	//dosilanie
	IF "DB10_instance_SCADA".actDTL_RechargingOn.HOUR < 0
	  OR "DB10_instance_SCADA".actDTL_RechargingOn.HOUR > 23
	  OR "dbHold_Sending".data."Time".Start_dosilanie_1.HOUR < 0
	  OR "dbHold_Sending".data."Time".Start_dosilanie_1.HOUR > 23
	THEN
	  // wypełnij zerami
	  "DB10_instance_SCADA".actDTL_RechargingOn.HOUR := 0;
	  "tempdbHold_SendingTCP".Start_dosilanie_1.HOUR := 0;
	  "dbHold_Sending".data."Time".Start_dosilanie_1.HOUR := 0;
	  ;
	END_IF;
	
	IF "DB10_instance_SCADA".actDTL_RechargingOn.MINUTE < 0
	  OR "DB10_instance_SCADA".actDTL_RechargingOn.MINUTE > 60
	  OR "dbHold_Sending".data."Time".Start_dosilanie_1.MINUTE < 0
	  OR "dbHold_Sending".data."Time".Start_dosilanie_1.MINUTE > 60
	THEN
	  // wypełnij zerami
	  "DB10_instance_SCADA".actDTL_RechargingOn.MINUTE := 0;
	  "tempdbHold_SendingTCP".Start_dosilanie_1.MINUTE := 0;
	  "dbHold_Sending".data."Time".Start_dosilanie_1.MINUTE := 0;
	  ;
	END_IF;
	
	// stop dosilanie
	IF "DB10_instance_SCADA".actDTL_RechargingOff.HOUR < 0
	  OR "DB10_instance_SCADA".actDTL_RechargingOff.HOUR > 23
	  OR "dbHold_Sending".data."Time".Stop_dosilanie_1.HOUR < 0
	  OR "dbHold_Sending".data."Time".Stop_dosilanie_1.HOUR > 23
	THEN
	  // wypełnij zerami
	  "DB10_instance_SCADA".actDTL_RechargingOff.HOUR := 0;
	  "tempdbHold_SendingTCP".Stop_dosilanie_1.HOUR := 0;
	  "dbHold_Sending".data."Time".Stop_dosilanie_1.HOUR := 0;
	  ;
	END_IF;
	
	IF "DB10_instance_SCADA".actDTL_RechargingOff.MINUTE < 0
	  OR "DB10_instance_SCADA".actDTL_RechargingOff.MINUTE > 60
	  OR "dbHold_Sending".data."Time".Stop_dosilanie_1.MINUTE < 0
	  OR "dbHold_Sending".data."Time".Stop_dosilanie_1.MINUTE > 60
	THEN
	  // wypełnij zerami
	  "DB10_instance_SCADA".actDTL_RechargingOff.MINUTE := 0;
	  "tempdbHold_SendingTCP".Stop_dosilanie_1.MINUTE := 0;
	  "dbHold_Sending".data."Time".Stop_dosilanie_1.MINUTE := 0;
	  ;
	END_IF;
	
	
	
	
	
	
	
END_FUNCTION

FUNCTION "Read_MPP04_2_ModbusRTU" : Void   // FC24, LAD
TITLE = Odczyt parametrów z MPP04 Pompownia / Read data from SC100
{ S7_Optimized_Access := 'TRUE' }
AUTHOR : rtecmer
VERSION : 0.1
// Czytanie z przepływomierza pompownia główna. Modbus RTU 19200, bit stop-1, parti-no
// Czytanie z SC1000 
// Obsługa protokołu Master Modbus RTU.  Odczyt pomiarów  i status czujnika SC1000
// stored: AutoNumber false, IsIECCheckEnabled false, SetENOAutomatically false, UDAEnableTagReadback false
   VAR_TEMP
      Wielkość_przeływu_Adres0_0 : DWord;
      Wielkość_przeływu_Adres0_1 : DWord;
      Wielkość_przeływu_Adres2_0 : DWord;
      Wielkość_przeływu_Adres2_2 : DWord;
   END_VAR
   VAR_TEMP   // added for the SCL form of the ladder/FBD networks
      _w1 : Bool;
      _w2 : Bool;
   END_VAR
BEGIN

REGION Network 1: Odczyt parametrów z MPP04 Studnia na tłocznym
   // Czytanie z przepływomierza pompownia główna. Modbus RTU 19200, bit stop-1, parti-no
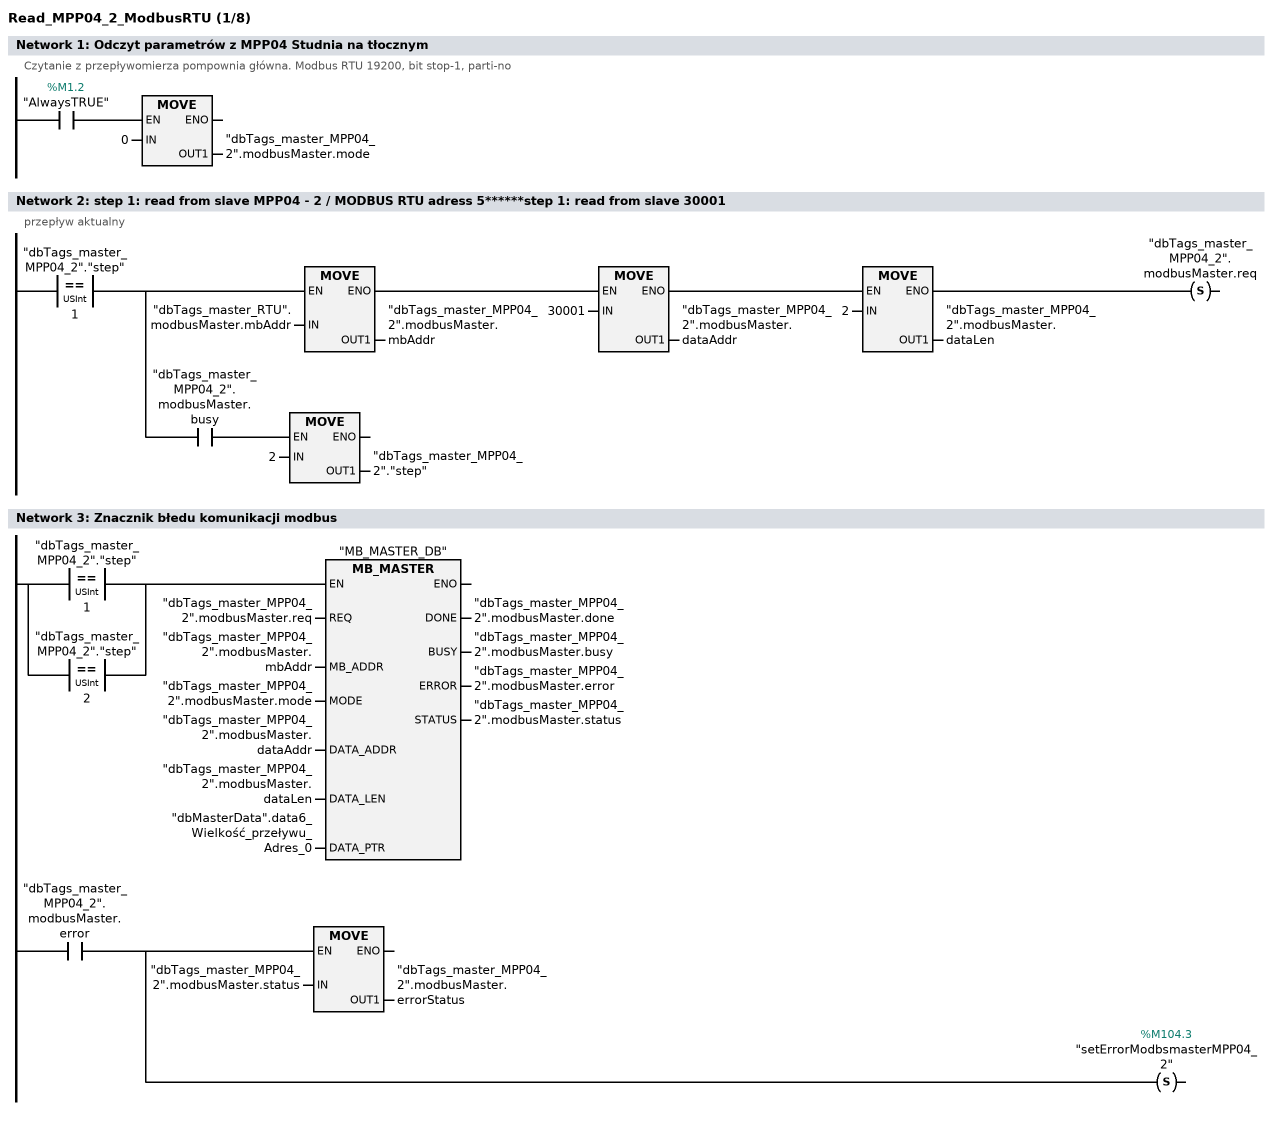
   RUNG wire#powerrail
      Contact( "AlwaysTRUE" )
      { S7_GenerateENO := "TRUE" } Move(in := 0, out1 => "dbTags_master_MPP04_2".modbusMaster.mode)
   END_RUNG
   // the same network as SCL:
   IF "AlwaysTRUE" THEN "dbTags_master_MPP04_2".modbusMaster.mode := 0; END_IF;
END_REGION

REGION Network 2: step 1: read from slave MPP04 - 2 / MODBUS RTU adress 5******step 1: read from slave 30001
   // przepływ aktualny
   RUNG wire#powerrail
      { S7_Templates := "SrcType := USInt" } EQ_Contact(in1 := "dbTags_master_MPP04_2"."step", in2 := 1)
      wire#w1
      Move(in := "dbTags_master_RTU".modbusMaster.mbAddr, out1 => "dbTags_master_MPP04_2".modbusMaster.mbAddr)
      { S7_GenerateENO := "TRUE" } Move(in := 30001, out1 => "dbTags_master_MPP04_2".modbusMaster.dataAddr)
      Move(in := 2, out1 => "dbTags_master_MPP04_2".modbusMaster.dataLen)
      S_Coil( "dbTags_master_MPP04_2".modbusMaster.req )
   END_RUNG
   RUNG wire#w1
      Contact( "dbTags_master_MPP04_2".modbusMaster.busy )
      { S7_GenerateENO := "TRUE" } Move(in := 2, out1 => "dbTags_master_MPP04_2"."step")
   END_RUNG
   // the same network as SCL:
   // ENO of a box is taken as its EN; it also drops when the box reports an error
   #_w1 := "dbTags_master_MPP04_2"."step" = 1;
   IF #_w1 THEN
       "dbTags_master_MPP04_2".modbusMaster.mbAddr := "dbTags_master_RTU".modbusMaster.mbAddr;
       "dbTags_master_MPP04_2".modbusMaster.dataAddr := 30001;
       "dbTags_master_MPP04_2".modbusMaster.dataLen := 2;
       "dbTags_master_MPP04_2".modbusMaster.req := TRUE;
   END_IF;
   IF #_w1 AND "dbTags_master_MPP04_2".modbusMaster.busy THEN "dbTags_master_MPP04_2"."step" := 2; END_IF;
END_REGION

REGION Network 3: Znacznik błedu komunikacji modbus
   RUNG wire#powerrail
      { S7_Templates := "SrcType := USInt" } EQ_Contact(in1 := "dbTags_master_MPP04_2"."step", in2 := 1)
      wire#w1
      "MB_MASTER_DB".MB_MASTER(REQ := "dbTags_master_MPP04_2".modbusMaster.req, MB_ADDR := "dbTags_master_MPP04_2".modbusMaster.mbAddr, MODE := "dbTags_master_MPP04_2".modbusMaster.mode, DATA_ADDR := "dbTags_master_MPP04_2".modbusMaster.dataAddr, DATA_LEN := "dbTags_master_MPP04_2".modbusMaster.dataLen, DATA_PTR := "dbMasterData".data6_Wielkość_przeływu_Adres_0, DONE => "dbTags_master_MPP04_2".modbusMaster.done, BUSY => "dbTags_master_MPP04_2".modbusMaster.busy, ERROR => "dbTags_master_MPP04_2".modbusMaster.error, STATUS => "dbTags_master_MPP04_2".modbusMaster.status)
   END_RUNG
   RUNG wire#powerrail
      { S7_Templates := "SrcType := USInt" } EQ_Contact(in1 := "dbTags_master_MPP04_2"."step", in2 := 2)
   END_RUNG wire#w1
   RUNG wire#powerrail
      Contact( "dbTags_master_MPP04_2".modbusMaster.error )
      wire#w2
      { S7_GenerateENO := "TRUE" } Move(in := "dbTags_master_MPP04_2".modbusMaster.status, out1 => "dbTags_master_MPP04_2".modbusMaster.errorStatus)
   END_RUNG
   RUNG wire#w2
      S_Coil( "setErrorModbsmasterMPP04_2" )
   END_RUNG
   // the same network as SCL:
   IF ("dbTags_master_MPP04_2"."step" = 1) OR ("dbTags_master_MPP04_2"."step" = 2) THEN
       "MB_MASTER_DB"(REQ := "dbTags_master_MPP04_2".modbusMaster.req,   // MB_MASTER
                      MB_ADDR := "dbTags_master_MPP04_2".modbusMaster.mbAddr,
                      MODE := "dbTags_master_MPP04_2".modbusMaster.mode,
                      DATA_ADDR := "dbTags_master_MPP04_2".modbusMaster.dataAddr,
                      DATA_LEN := "dbTags_master_MPP04_2".modbusMaster.dataLen,
                      DATA_PTR := "dbMasterData".data6_Wielkość_przeływu_Adres_0,
                      DONE => "dbTags_master_MPP04_2".modbusMaster.done,
                      BUSY => "dbTags_master_MPP04_2".modbusMaster.busy,
                      ERROR => "dbTags_master_MPP04_2".modbusMaster.error,
                      STATUS => "dbTags_master_MPP04_2".modbusMaster.status);
   END_IF;
   IF "dbTags_master_MPP04_2".modbusMaster.error THEN
       "dbTags_master_MPP04_2".modbusMaster.errorStatus := "dbTags_master_MPP04_2".modbusMaster.status;
       "setErrorModbsmasterMPP04_2" := TRUE;
   END_IF;
END_REGION

REGION Network 4: step 4: save received data / step 2: save received data 30001
   // Pomiar Temperatury KDN1
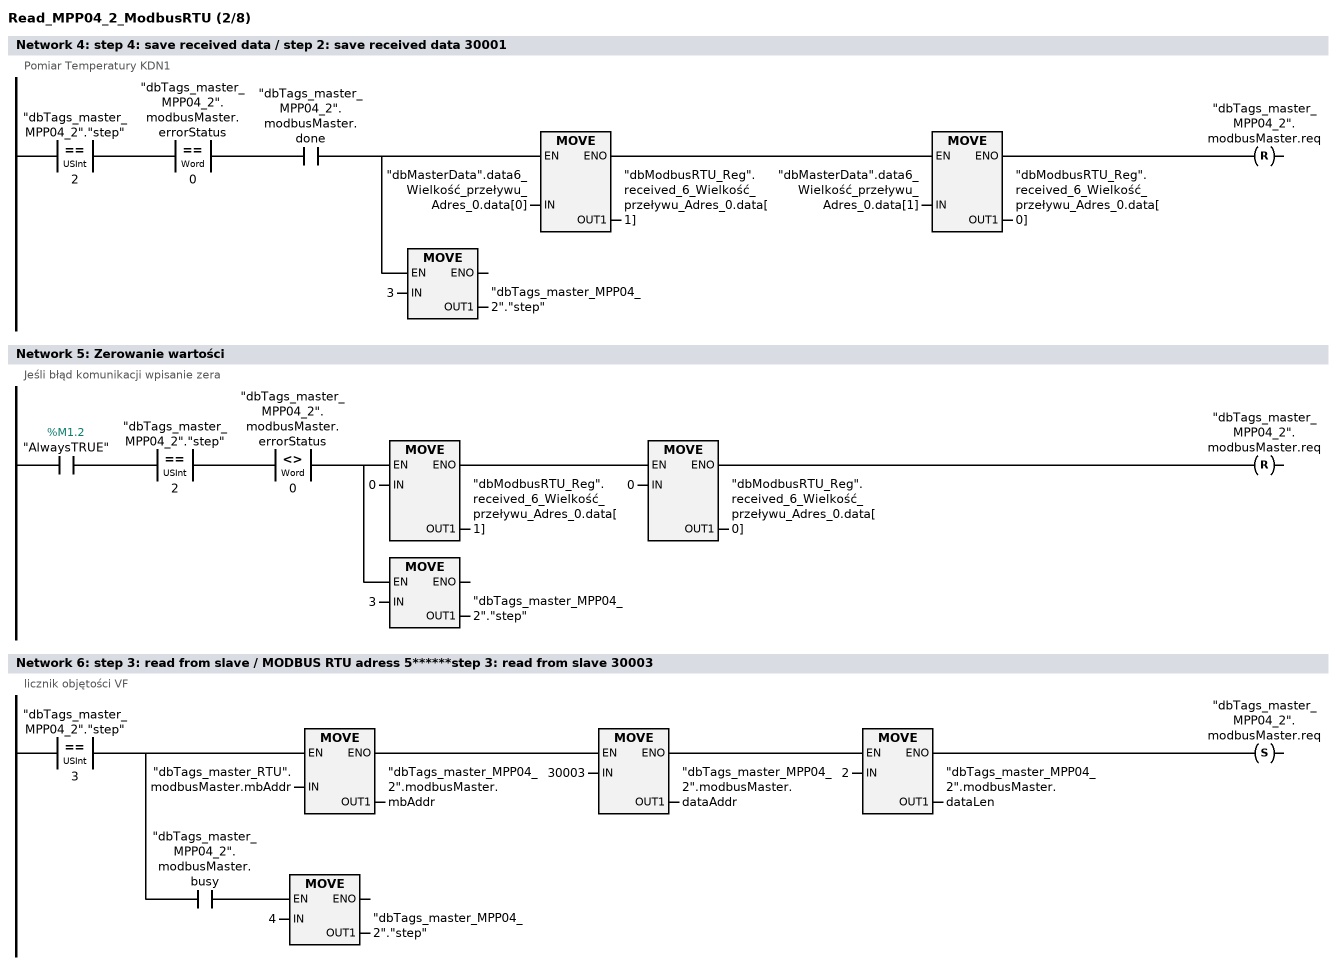
   RUNG wire#powerrail
      { S7_Templates := "SrcType := USInt" } EQ_Contact(in1 := "dbTags_master_MPP04_2"."step", in2 := 2)
      { S7_Templates := "SrcType := Word" } EQ_Contact(in1 := "dbTags_master_MPP04_2".modbusMaster.errorStatus, in2 := 0)
      Contact( "dbTags_master_MPP04_2".modbusMaster.done )
      wire#w1
      { S7_GenerateENO := "TRUE" } Move(in := "dbMasterData".data6_Wielkość_przeływu_Adres_0.data[0], out1 => "dbModbusRTU_Reg".received_6_Wielkość_przeływu_Adres_0.data[1])
      { S7_GenerateENO := "TRUE" } Move(in := "dbMasterData".data6_Wielkość_przeływu_Adres_0.data[1], out1 => "dbModbusRTU_Reg".received_6_Wielkość_przeływu_Adres_0.data[0])
      R_Coil( "dbTags_master_MPP04_2".modbusMaster.req )
   END_RUNG
   RUNG wire#w1
      { S7_GenerateENO := "TRUE" } Move(in := 3, out1 => "dbTags_master_MPP04_2"."step")
   END_RUNG
   // the same network as SCL:
   // ENO of a box is taken as its EN; it also drops when the box reports an error
   IF ("dbTags_master_MPP04_2"."step" = 2) AND ("dbTags_master_MPP04_2".modbusMaster.errorStatus = 0) AND "dbTags_master_MPP04_2".modbusMaster.done THEN
       "dbModbusRTU_Reg".received_6_Wielkość_przeływu_Adres_0.data[1] := "dbMasterData".data6_Wielkość_przeływu_Adres_0.data[0];
       "dbModbusRTU_Reg".received_6_Wielkość_przeływu_Adres_0.data[0] := "dbMasterData".data6_Wielkość_przeływu_Adres_0.data[1];
       "dbTags_master_MPP04_2".modbusMaster.req := FALSE;
       "dbTags_master_MPP04_2"."step" := 3;
   END_IF;
END_REGION

REGION Network 5: Zerowanie wartości
   // Jeśli błąd komunikacji wpisanie zera
   RUNG wire#powerrail
      Contact( "AlwaysTRUE" )
      { S7_Templates := "SrcType := USInt" } EQ_Contact(in1 := "dbTags_master_MPP04_2"."step", in2 := 2)
      { S7_Templates := "SrcType := Word" } NE_Contact(in1 := "dbTags_master_MPP04_2".modbusMaster.errorStatus, in2 := 0)
      wire#w1
      { S7_GenerateENO := "TRUE" } Move(in := 0, out1 => "dbModbusRTU_Reg".received_6_Wielkość_przeływu_Adres_0.data[1])
      { S7_GenerateENO := "TRUE" } Move(in := 0, out1 => "dbModbusRTU_Reg".received_6_Wielkość_przeływu_Adres_0.data[0])
      R_Coil( "dbTags_master_MPP04_2".modbusMaster.req )
   END_RUNG
   RUNG wire#w1
      { S7_GenerateENO := "TRUE" } Move(in := 3, out1 => "dbTags_master_MPP04_2"."step")
   END_RUNG
   // the same network as SCL:
   // ENO of a box is taken as its EN; it also drops when the box reports an error
   IF "AlwaysTRUE" AND ("dbTags_master_MPP04_2"."step" = 2) AND ("dbTags_master_MPP04_2".modbusMaster.errorStatus <> 0) THEN
       "dbModbusRTU_Reg".received_6_Wielkość_przeływu_Adres_0.data[1] := 0;
       "dbModbusRTU_Reg".received_6_Wielkość_przeływu_Adres_0.data[0] := 0;
       "dbTags_master_MPP04_2".modbusMaster.req := FALSE;
       "dbTags_master_MPP04_2"."step" := 3;
   END_IF;
END_REGION

REGION Network 6: step 3: read from slave / MODBUS RTU adress 5******step 3: read from slave 30003
   // licznik objętości VF
   RUNG wire#powerrail
      { S7_Templates := "SrcType := USInt" } EQ_Contact(in1 := "dbTags_master_MPP04_2"."step", in2 := 3)
      wire#w1
      Move(in := "dbTags_master_RTU".modbusMaster.mbAddr, out1 => "dbTags_master_MPP04_2".modbusMaster.mbAddr)
      { S7_GenerateENO := "TRUE" } Move(in := 30003, out1 => "dbTags_master_MPP04_2".modbusMaster.dataAddr)
      Move(in := 2, out1 => "dbTags_master_MPP04_2".modbusMaster.dataLen)
      S_Coil( "dbTags_master_MPP04_2".modbusMaster.req )
   END_RUNG
   RUNG wire#w1
      Contact( "dbTags_master_MPP04_2".modbusMaster.busy )
      { S7_GenerateENO := "TRUE" } Move(in := 4, out1 => "dbTags_master_MPP04_2"."step")
   END_RUNG
   // the same network as SCL:
   // ENO of a box is taken as its EN; it also drops when the box reports an error
   #_w1 := "dbTags_master_MPP04_2"."step" = 3;
   IF #_w1 THEN
       "dbTags_master_MPP04_2".modbusMaster.mbAddr := "dbTags_master_RTU".modbusMaster.mbAddr;
       "dbTags_master_MPP04_2".modbusMaster.dataAddr := 30003;
       "dbTags_master_MPP04_2".modbusMaster.dataLen := 2;
       "dbTags_master_MPP04_2".modbusMaster.req := TRUE;
   END_IF;
   IF #_w1 AND "dbTags_master_MPP04_2".modbusMaster.busy THEN "dbTags_master_MPP04_2"."step" := 4; END_IF;
END_REGION

REGION Network 7: Znacznik błedu komunikacji modbus
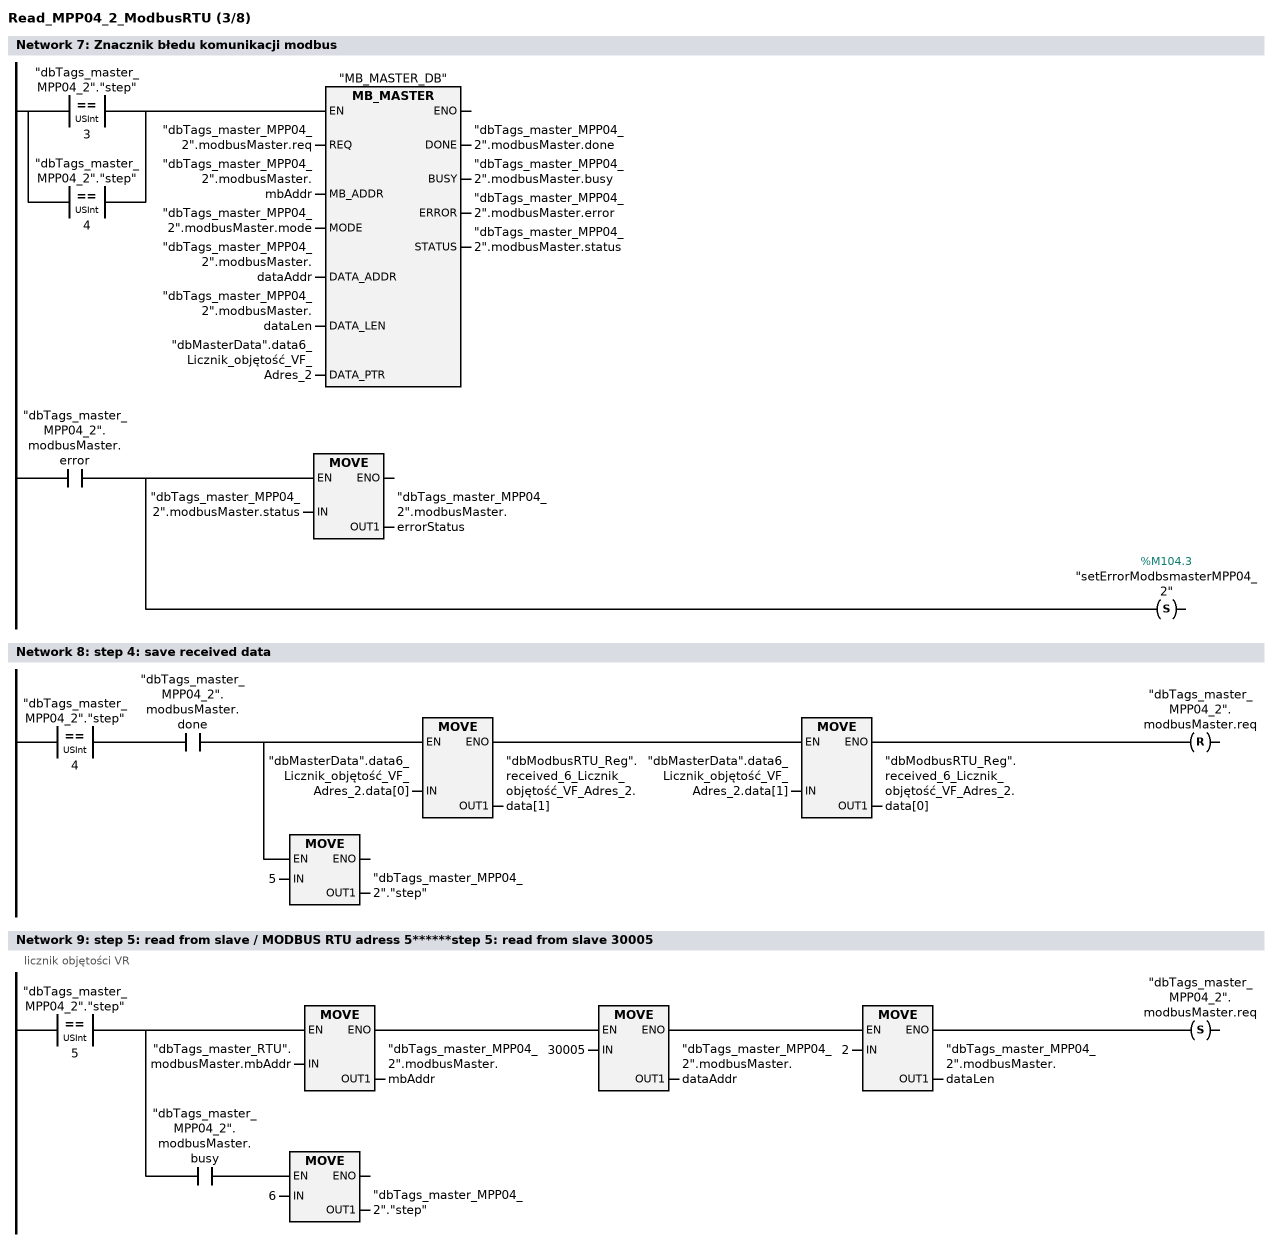
   RUNG wire#powerrail
      { S7_Templates := "SrcType := USInt" } EQ_Contact(in1 := "dbTags_master_MPP04_2"."step", in2 := 3)
      wire#w1
      "MB_MASTER_DB".MB_MASTER(REQ := "dbTags_master_MPP04_2".modbusMaster.req, MB_ADDR := "dbTags_master_MPP04_2".modbusMaster.mbAddr, MODE := "dbTags_master_MPP04_2".modbusMaster.mode, DATA_ADDR := "dbTags_master_MPP04_2".modbusMaster.dataAddr, DATA_LEN := "dbTags_master_MPP04_2".modbusMaster.dataLen, DATA_PTR := "dbMasterData".data6_Licznik_objętość_VF_Adres_2, DONE => "dbTags_master_MPP04_2".modbusMaster.done, BUSY => "dbTags_master_MPP04_2".modbusMaster.busy, ERROR => "dbTags_master_MPP04_2".modbusMaster.error, STATUS => "dbTags_master_MPP04_2".modbusMaster.status)
   END_RUNG
   RUNG wire#powerrail
      { S7_Templates := "SrcType := USInt" } EQ_Contact(in1 := "dbTags_master_MPP04_2"."step", in2 := 4)
   END_RUNG wire#w1
   RUNG wire#powerrail
      Contact( "dbTags_master_MPP04_2".modbusMaster.error )
      wire#w2
      { S7_GenerateENO := "TRUE" } Move(in := "dbTags_master_MPP04_2".modbusMaster.status, out1 => "dbTags_master_MPP04_2".modbusMaster.errorStatus)
   END_RUNG
   RUNG wire#w2
      S_Coil( "setErrorModbsmasterMPP04_2" )
   END_RUNG
   // the same network as SCL:
   IF ("dbTags_master_MPP04_2"."step" = 3) OR ("dbTags_master_MPP04_2"."step" = 4) THEN
       "MB_MASTER_DB"(REQ := "dbTags_master_MPP04_2".modbusMaster.req,   // MB_MASTER
                      MB_ADDR := "dbTags_master_MPP04_2".modbusMaster.mbAddr,
                      MODE := "dbTags_master_MPP04_2".modbusMaster.mode,
                      DATA_ADDR := "dbTags_master_MPP04_2".modbusMaster.dataAddr,
                      DATA_LEN := "dbTags_master_MPP04_2".modbusMaster.dataLen,
                      DATA_PTR := "dbMasterData".data6_Licznik_objętość_VF_Adres_2,
                      DONE => "dbTags_master_MPP04_2".modbusMaster.done,
                      BUSY => "dbTags_master_MPP04_2".modbusMaster.busy,
                      ERROR => "dbTags_master_MPP04_2".modbusMaster.error,
                      STATUS => "dbTags_master_MPP04_2".modbusMaster.status);
   END_IF;
   IF "dbTags_master_MPP04_2".modbusMaster.error THEN
       "dbTags_master_MPP04_2".modbusMaster.errorStatus := "dbTags_master_MPP04_2".modbusMaster.status;
       "setErrorModbsmasterMPP04_2" := TRUE;
   END_IF;
END_REGION

REGION Network 8: step 4: save received data
   RUNG wire#powerrail
      { S7_Templates := "SrcType := USInt" } EQ_Contact(in1 := "dbTags_master_MPP04_2"."step", in2 := 4)
      Contact( "dbTags_master_MPP04_2".modbusMaster.done )
      wire#w1
      { S7_GenerateENO := "TRUE" } Move(in := "dbMasterData".data6_Licznik_objętość_VF_Adres_2.data[0], out1 => "dbModbusRTU_Reg".received_6_Licznik_objętość_VF_Adres_2.data[1])
      { S7_GenerateENO := "TRUE" } Move(in := "dbMasterData".data6_Licznik_objętość_VF_Adres_2.data[1], out1 => "dbModbusRTU_Reg".received_6_Licznik_objętość_VF_Adres_2.data[0])
      R_Coil( "dbTags_master_MPP04_2".modbusMaster.req )
   END_RUNG
   RUNG wire#w1
      { S7_GenerateENO := "TRUE" } Move(in := 5, out1 => "dbTags_master_MPP04_2"."step")
   END_RUNG
   // the same network as SCL:
   // ENO of a box is taken as its EN; it also drops when the box reports an error
   IF ("dbTags_master_MPP04_2"."step" = 4) AND "dbTags_master_MPP04_2".modbusMaster.done THEN
       "dbModbusRTU_Reg".received_6_Licznik_objętość_VF_Adres_2.data[1] := "dbMasterData".data6_Licznik_objętość_VF_Adres_2.data[0];
       "dbModbusRTU_Reg".received_6_Licznik_objętość_VF_Adres_2.data[0] := "dbMasterData".data6_Licznik_objętość_VF_Adres_2.data[1];
       "dbTags_master_MPP04_2".modbusMaster.req := FALSE;
       "dbTags_master_MPP04_2"."step" := 5;
   END_IF;
END_REGION

REGION Network 9: step 5: read from slave / MODBUS RTU adress 5******step 5: read from slave 30005
   // licznik objętości VR
   RUNG wire#powerrail
      { S7_Templates := "SrcType := USInt" } EQ_Contact(in1 := "dbTags_master_MPP04_2"."step", in2 := 5)
      wire#w1
      Move(in := "dbTags_master_RTU".modbusMaster.mbAddr, out1 => "dbTags_master_MPP04_2".modbusMaster.mbAddr)
      { S7_GenerateENO := "TRUE" } Move(in := 30005, out1 => "dbTags_master_MPP04_2".modbusMaster.dataAddr)
      Move(in := 2, out1 => "dbTags_master_MPP04_2".modbusMaster.dataLen)
      S_Coil( "dbTags_master_MPP04_2".modbusMaster.req )
   END_RUNG
   RUNG wire#w1
      Contact( "dbTags_master_MPP04_2".modbusMaster.busy )
      { S7_GenerateENO := "TRUE" } Move(in := 6, out1 => "dbTags_master_MPP04_2"."step")
   END_RUNG
   // the same network as SCL:
   // ENO of a box is taken as its EN; it also drops when the box reports an error
   #_w1 := "dbTags_master_MPP04_2"."step" = 5;
   IF #_w1 THEN
       "dbTags_master_MPP04_2".modbusMaster.mbAddr := "dbTags_master_RTU".modbusMaster.mbAddr;
       "dbTags_master_MPP04_2".modbusMaster.dataAddr := 30005;
       "dbTags_master_MPP04_2".modbusMaster.dataLen := 2;
       "dbTags_master_MPP04_2".modbusMaster.req := TRUE;
   END_IF;
   IF #_w1 AND "dbTags_master_MPP04_2".modbusMaster.busy THEN "dbTags_master_MPP04_2"."step" := 6; END_IF;
END_REGION

REGION Network 10: Znacznik błedu komunikacji modbus
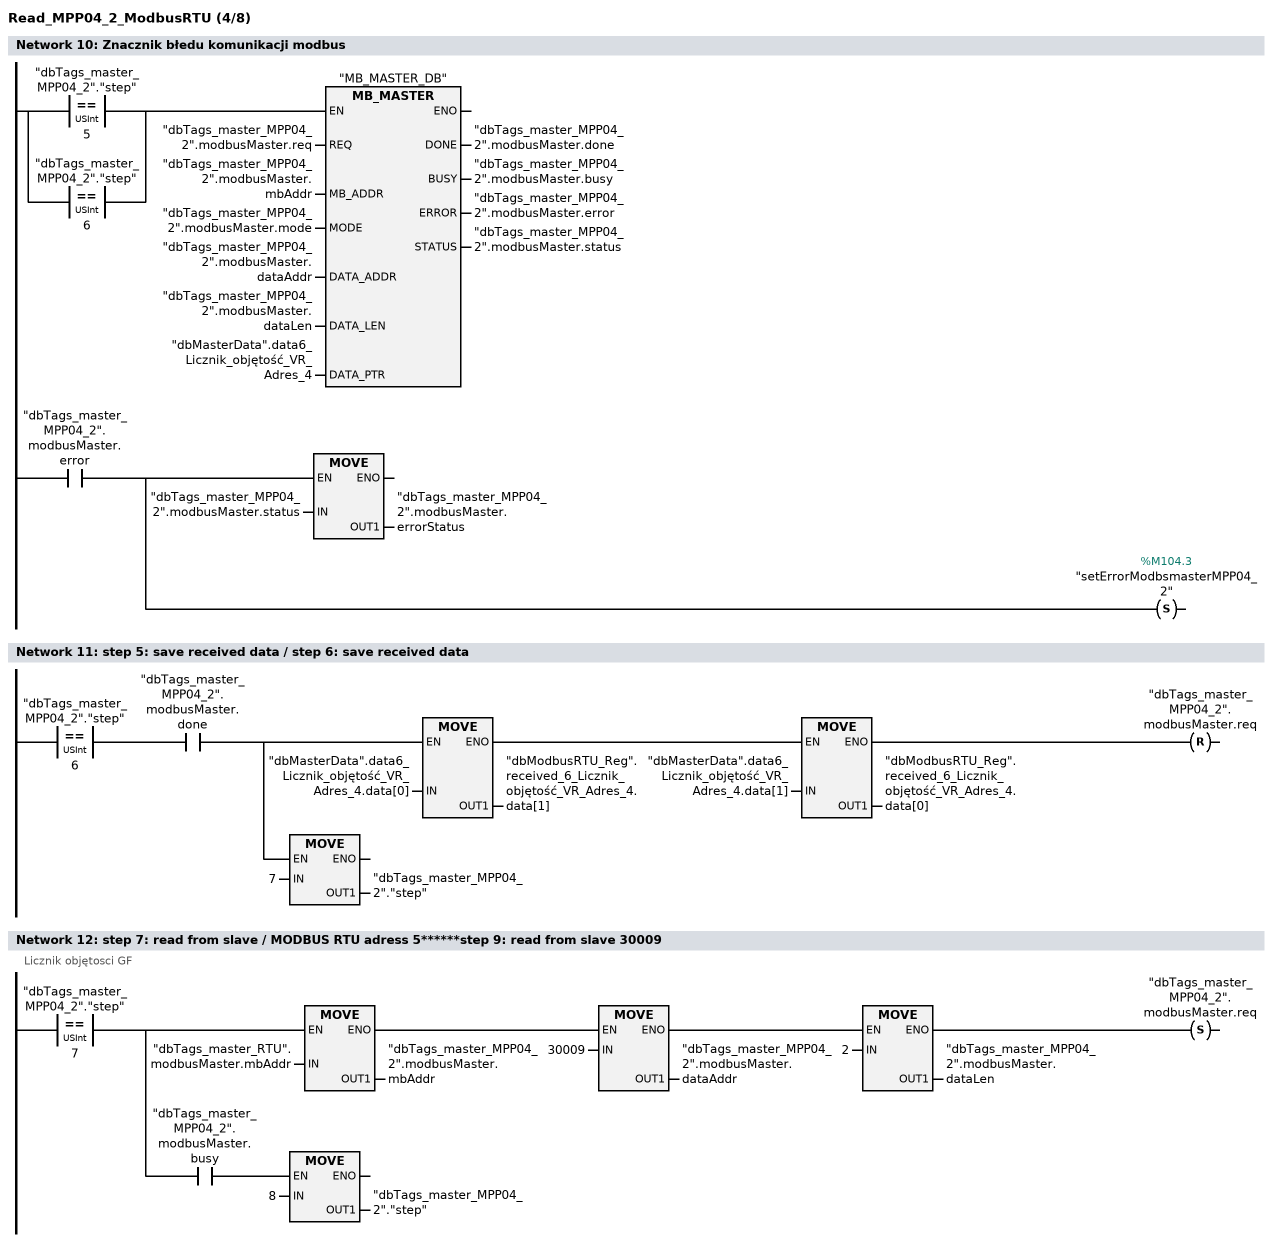
   RUNG wire#powerrail
      { S7_Templates := "SrcType := USInt" } EQ_Contact(in1 := "dbTags_master_MPP04_2"."step", in2 := 5)
      wire#w1
      "MB_MASTER_DB".MB_MASTER(REQ := "dbTags_master_MPP04_2".modbusMaster.req, MB_ADDR := "dbTags_master_MPP04_2".modbusMaster.mbAddr, MODE := "dbTags_master_MPP04_2".modbusMaster.mode, DATA_ADDR := "dbTags_master_MPP04_2".modbusMaster.dataAddr, DATA_LEN := "dbTags_master_MPP04_2".modbusMaster.dataLen, DATA_PTR := "dbMasterData".data6_Licznik_objętość_VR_Adres_4, DONE => "dbTags_master_MPP04_2".modbusMaster.done, BUSY => "dbTags_master_MPP04_2".modbusMaster.busy, ERROR => "dbTags_master_MPP04_2".modbusMaster.error, STATUS => "dbTags_master_MPP04_2".modbusMaster.status)
   END_RUNG
   RUNG wire#powerrail
      { S7_Templates := "SrcType := USInt" } EQ_Contact(in1 := "dbTags_master_MPP04_2"."step", in2 := 6)
   END_RUNG wire#w1
   RUNG wire#powerrail
      Contact( "dbTags_master_MPP04_2".modbusMaster.error )
      wire#w2
      { S7_GenerateENO := "TRUE" } Move(in := "dbTags_master_MPP04_2".modbusMaster.status, out1 => "dbTags_master_MPP04_2".modbusMaster.errorStatus)
   END_RUNG
   RUNG wire#w2
      S_Coil( "setErrorModbsmasterMPP04_2" )
   END_RUNG
   // the same network as SCL:
   IF ("dbTags_master_MPP04_2"."step" = 5) OR ("dbTags_master_MPP04_2"."step" = 6) THEN
       "MB_MASTER_DB"(REQ := "dbTags_master_MPP04_2".modbusMaster.req,   // MB_MASTER
                      MB_ADDR := "dbTags_master_MPP04_2".modbusMaster.mbAddr,
                      MODE := "dbTags_master_MPP04_2".modbusMaster.mode,
                      DATA_ADDR := "dbTags_master_MPP04_2".modbusMaster.dataAddr,
                      DATA_LEN := "dbTags_master_MPP04_2".modbusMaster.dataLen,
                      DATA_PTR := "dbMasterData".data6_Licznik_objętość_VR_Adres_4,
                      DONE => "dbTags_master_MPP04_2".modbusMaster.done,
                      BUSY => "dbTags_master_MPP04_2".modbusMaster.busy,
                      ERROR => "dbTags_master_MPP04_2".modbusMaster.error,
                      STATUS => "dbTags_master_MPP04_2".modbusMaster.status);
   END_IF;
   IF "dbTags_master_MPP04_2".modbusMaster.error THEN
       "dbTags_master_MPP04_2".modbusMaster.errorStatus := "dbTags_master_MPP04_2".modbusMaster.status;
       "setErrorModbsmasterMPP04_2" := TRUE;
   END_IF;
END_REGION

REGION Network 11: step 5: save received data / step 6: save received data
   RUNG wire#powerrail
      { S7_Templates := "SrcType := USInt" } EQ_Contact(in1 := "dbTags_master_MPP04_2"."step", in2 := 6)
      Contact( "dbTags_master_MPP04_2".modbusMaster.done )
      wire#w1
      { S7_GenerateENO := "TRUE" } Move(in := "dbMasterData".data6_Licznik_objętość_VR_Adres_4.data[0], out1 => "dbModbusRTU_Reg".received_6_Licznik_objętość_VR_Adres_4.data[1])
      { S7_GenerateENO := "TRUE" } Move(in := "dbMasterData".data6_Licznik_objętość_VR_Adres_4.data[1], out1 => "dbModbusRTU_Reg".received_6_Licznik_objętość_VR_Adres_4.data[0])
      R_Coil( "dbTags_master_MPP04_2".modbusMaster.req )
   END_RUNG
   RUNG wire#w1
      { S7_GenerateENO := "TRUE" } Move(in := 7, out1 => "dbTags_master_MPP04_2"."step")
   END_RUNG
   // the same network as SCL:
   // ENO of a box is taken as its EN; it also drops when the box reports an error
   IF ("dbTags_master_MPP04_2"."step" = 6) AND "dbTags_master_MPP04_2".modbusMaster.done THEN
       "dbModbusRTU_Reg".received_6_Licznik_objętość_VR_Adres_4.data[1] := "dbMasterData".data6_Licznik_objętość_VR_Adres_4.data[0];
       "dbModbusRTU_Reg".received_6_Licznik_objętość_VR_Adres_4.data[0] := "dbMasterData".data6_Licznik_objętość_VR_Adres_4.data[1];
       "dbTags_master_MPP04_2".modbusMaster.req := FALSE;
       "dbTags_master_MPP04_2"."step" := 7;
   END_IF;
END_REGION

REGION Network 12: step 7: read from slave / MODBUS RTU adress 5******step 9: read from slave 30009
   // Licznik objętosci GF
   RUNG wire#powerrail
      { S7_Templates := "SrcType := USInt" } EQ_Contact(in1 := "dbTags_master_MPP04_2"."step", in2 := 7)
      wire#w1
      Move(in := "dbTags_master_RTU".modbusMaster.mbAddr, out1 => "dbTags_master_MPP04_2".modbusMaster.mbAddr)
      { S7_GenerateENO := "TRUE" } Move(in := 30009, out1 => "dbTags_master_MPP04_2".modbusMaster.dataAddr)
      Move(in := 2, out1 => "dbTags_master_MPP04_2".modbusMaster.dataLen)
      S_Coil( "dbTags_master_MPP04_2".modbusMaster.req )
   END_RUNG
   RUNG wire#w1
      Contact( "dbTags_master_MPP04_2".modbusMaster.busy )
      { S7_GenerateENO := "TRUE" } Move(in := 8, out1 => "dbTags_master_MPP04_2"."step")
   END_RUNG
   // the same network as SCL:
   // ENO of a box is taken as its EN; it also drops when the box reports an error
   #_w1 := "dbTags_master_MPP04_2"."step" = 7;
   IF #_w1 THEN
       "dbTags_master_MPP04_2".modbusMaster.mbAddr := "dbTags_master_RTU".modbusMaster.mbAddr;
       "dbTags_master_MPP04_2".modbusMaster.dataAddr := 30009;
       "dbTags_master_MPP04_2".modbusMaster.dataLen := 2;
       "dbTags_master_MPP04_2".modbusMaster.req := TRUE;
   END_IF;
   IF #_w1 AND "dbTags_master_MPP04_2".modbusMaster.busy THEN "dbTags_master_MPP04_2"."step" := 8; END_IF;
END_REGION

REGION Network 13: Znacznik błedu komunikacji modbus
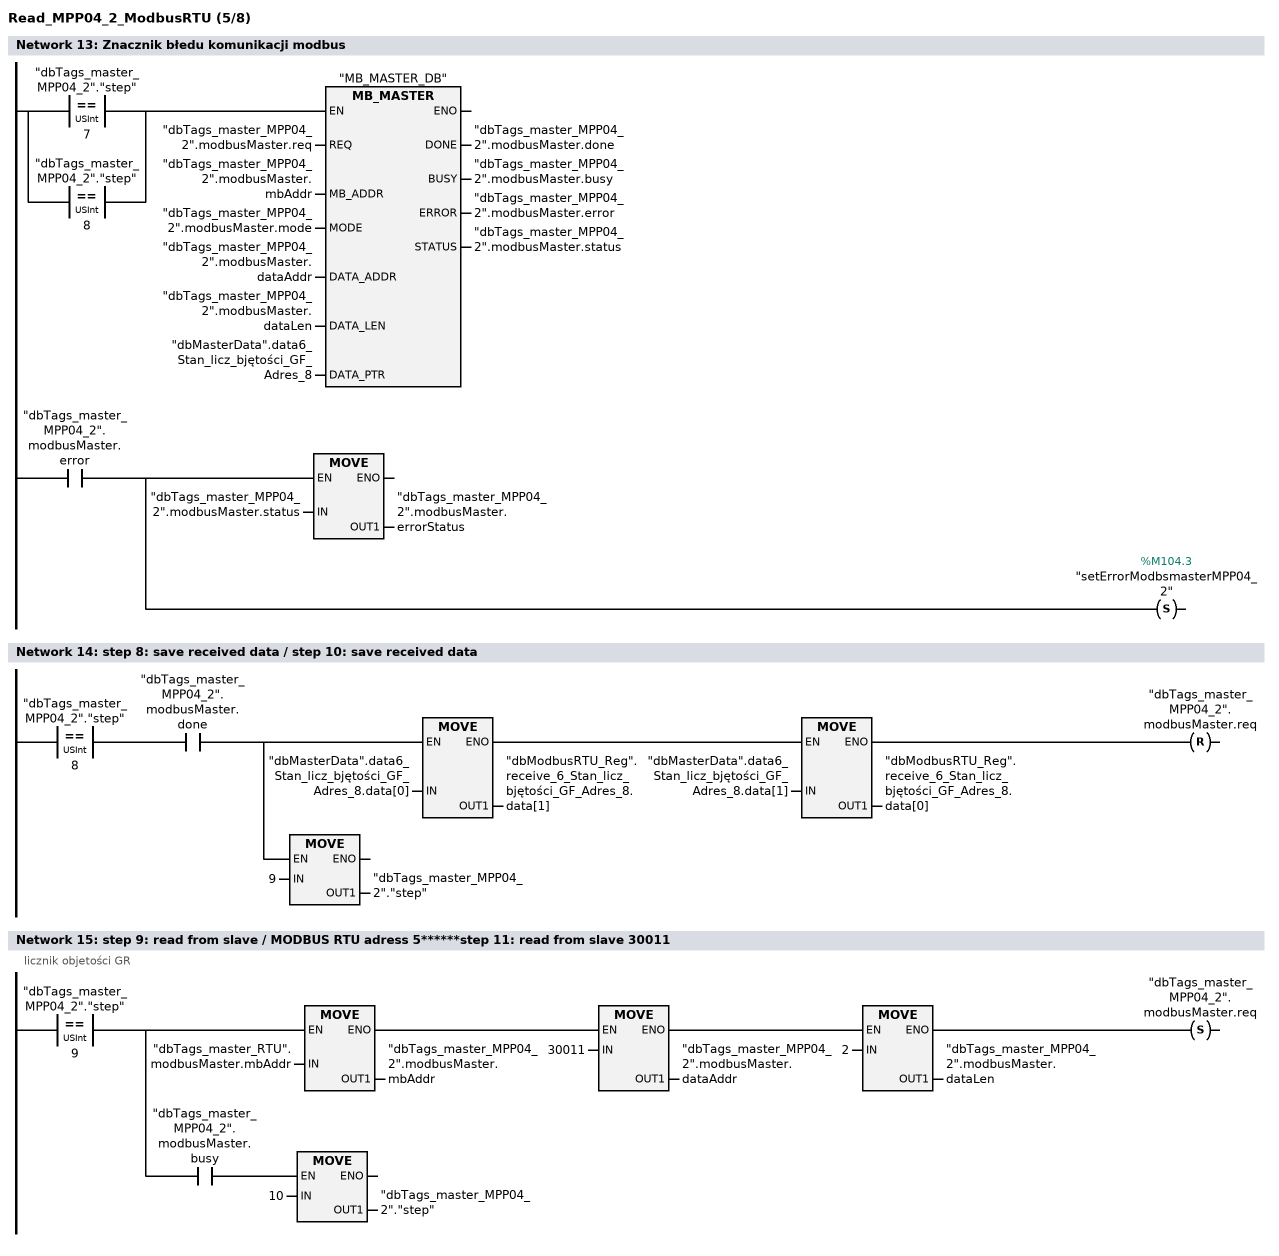
   RUNG wire#powerrail
      { S7_Templates := "SrcType := USInt" } EQ_Contact(in1 := "dbTags_master_MPP04_2"."step", in2 := 7)
      wire#w1
      "MB_MASTER_DB".MB_MASTER(REQ := "dbTags_master_MPP04_2".modbusMaster.req, MB_ADDR := "dbTags_master_MPP04_2".modbusMaster.mbAddr, MODE := "dbTags_master_MPP04_2".modbusMaster.mode, DATA_ADDR := "dbTags_master_MPP04_2".modbusMaster.dataAddr, DATA_LEN := "dbTags_master_MPP04_2".modbusMaster.dataLen, DATA_PTR := "dbMasterData".data6_Stan_licz_bjętości_GF_Adres_8, DONE => "dbTags_master_MPP04_2".modbusMaster.done, BUSY => "dbTags_master_MPP04_2".modbusMaster.busy, ERROR => "dbTags_master_MPP04_2".modbusMaster.error, STATUS => "dbTags_master_MPP04_2".modbusMaster.status)
   END_RUNG
   RUNG wire#powerrail
      { S7_Templates := "SrcType := USInt" } EQ_Contact(in1 := "dbTags_master_MPP04_2"."step", in2 := 8)
   END_RUNG wire#w1
   RUNG wire#powerrail
      Contact( "dbTags_master_MPP04_2".modbusMaster.error )
      wire#w2
      { S7_GenerateENO := "TRUE" } Move(in := "dbTags_master_MPP04_2".modbusMaster.status, out1 => "dbTags_master_MPP04_2".modbusMaster.errorStatus)
   END_RUNG
   RUNG wire#w2
      S_Coil( "setErrorModbsmasterMPP04_2" )
   END_RUNG
   // the same network as SCL:
   IF ("dbTags_master_MPP04_2"."step" = 7) OR ("dbTags_master_MPP04_2"."step" = 8) THEN
       "MB_MASTER_DB"(REQ := "dbTags_master_MPP04_2".modbusMaster.req,   // MB_MASTER
                      MB_ADDR := "dbTags_master_MPP04_2".modbusMaster.mbAddr,
                      MODE := "dbTags_master_MPP04_2".modbusMaster.mode,
                      DATA_ADDR := "dbTags_master_MPP04_2".modbusMaster.dataAddr,
                      DATA_LEN := "dbTags_master_MPP04_2".modbusMaster.dataLen,
                      DATA_PTR := "dbMasterData".data6_Stan_licz_bjętości_GF_Adres_8,
                      DONE => "dbTags_master_MPP04_2".modbusMaster.done,
                      BUSY => "dbTags_master_MPP04_2".modbusMaster.busy,
                      ERROR => "dbTags_master_MPP04_2".modbusMaster.error,
                      STATUS => "dbTags_master_MPP04_2".modbusMaster.status);
   END_IF;
   IF "dbTags_master_MPP04_2".modbusMaster.error THEN
       "dbTags_master_MPP04_2".modbusMaster.errorStatus := "dbTags_master_MPP04_2".modbusMaster.status;
       "setErrorModbsmasterMPP04_2" := TRUE;
   END_IF;
END_REGION

REGION Network 14: step 8: save received data / step 10: save received data
   RUNG wire#powerrail
      { S7_Templates := "SrcType := USInt" } EQ_Contact(in1 := "dbTags_master_MPP04_2"."step", in2 := 8)
      Contact( "dbTags_master_MPP04_2".modbusMaster.done )
      wire#w1
      { S7_GenerateENO := "TRUE" } Move(in := "dbMasterData".data6_Stan_licz_bjętości_GF_Adres_8.data[0], out1 => "dbModbusRTU_Reg".receive_6_Stan_licz_bjętości_GF_Adres_8.data[1])
      { S7_GenerateENO := "TRUE" } Move(in := "dbMasterData".data6_Stan_licz_bjętości_GF_Adres_8.data[1], out1 => "dbModbusRTU_Reg".receive_6_Stan_licz_bjętości_GF_Adres_8.data[0])
      R_Coil( "dbTags_master_MPP04_2".modbusMaster.req )
   END_RUNG
   RUNG wire#w1
      { S7_GenerateENO := "TRUE" } Move(in := 9, out1 => "dbTags_master_MPP04_2"."step")
   END_RUNG
   // the same network as SCL:
   // ENO of a box is taken as its EN; it also drops when the box reports an error
   IF ("dbTags_master_MPP04_2"."step" = 8) AND "dbTags_master_MPP04_2".modbusMaster.done THEN
       "dbModbusRTU_Reg".receive_6_Stan_licz_bjętości_GF_Adres_8.data[1] := "dbMasterData".data6_Stan_licz_bjętości_GF_Adres_8.data[0];
       "dbModbusRTU_Reg".receive_6_Stan_licz_bjętości_GF_Adres_8.data[0] := "dbMasterData".data6_Stan_licz_bjętości_GF_Adres_8.data[1];
       "dbTags_master_MPP04_2".modbusMaster.req := FALSE;
       "dbTags_master_MPP04_2"."step" := 9;
   END_IF;
END_REGION

REGION Network 15: step 9: read from slave / MODBUS RTU adress 5******step 11: read from slave 30011
   // licznik objetości GR
   RUNG wire#powerrail
      { S7_Templates := "SrcType := USInt" } EQ_Contact(in1 := "dbTags_master_MPP04_2"."step", in2 := 9)
      wire#w1
      Move(in := "dbTags_master_RTU".modbusMaster.mbAddr, out1 => "dbTags_master_MPP04_2".modbusMaster.mbAddr)
      { S7_GenerateENO := "TRUE" } Move(in := 30011, out1 => "dbTags_master_MPP04_2".modbusMaster.dataAddr)
      Move(in := 2, out1 => "dbTags_master_MPP04_2".modbusMaster.dataLen)
      S_Coil( "dbTags_master_MPP04_2".modbusMaster.req )
   END_RUNG
   RUNG wire#w1
      Contact( "dbTags_master_MPP04_2".modbusMaster.busy )
      { S7_GenerateENO := "TRUE" } Move(in := 10, out1 => "dbTags_master_MPP04_2"."step")
   END_RUNG
   // the same network as SCL:
   // ENO of a box is taken as its EN; it also drops when the box reports an error
   #_w1 := "dbTags_master_MPP04_2"."step" = 9;
   IF #_w1 THEN
       "dbTags_master_MPP04_2".modbusMaster.mbAddr := "dbTags_master_RTU".modbusMaster.mbAddr;
       "dbTags_master_MPP04_2".modbusMaster.dataAddr := 30011;
       "dbTags_master_MPP04_2".modbusMaster.dataLen := 2;
       "dbTags_master_MPP04_2".modbusMaster.req := TRUE;
   END_IF;
   IF #_w1 AND "dbTags_master_MPP04_2".modbusMaster.busy THEN "dbTags_master_MPP04_2"."step" := 10; END_IF;
END_REGION

REGION Network 16: Znacznik błedu komunikacji modbus
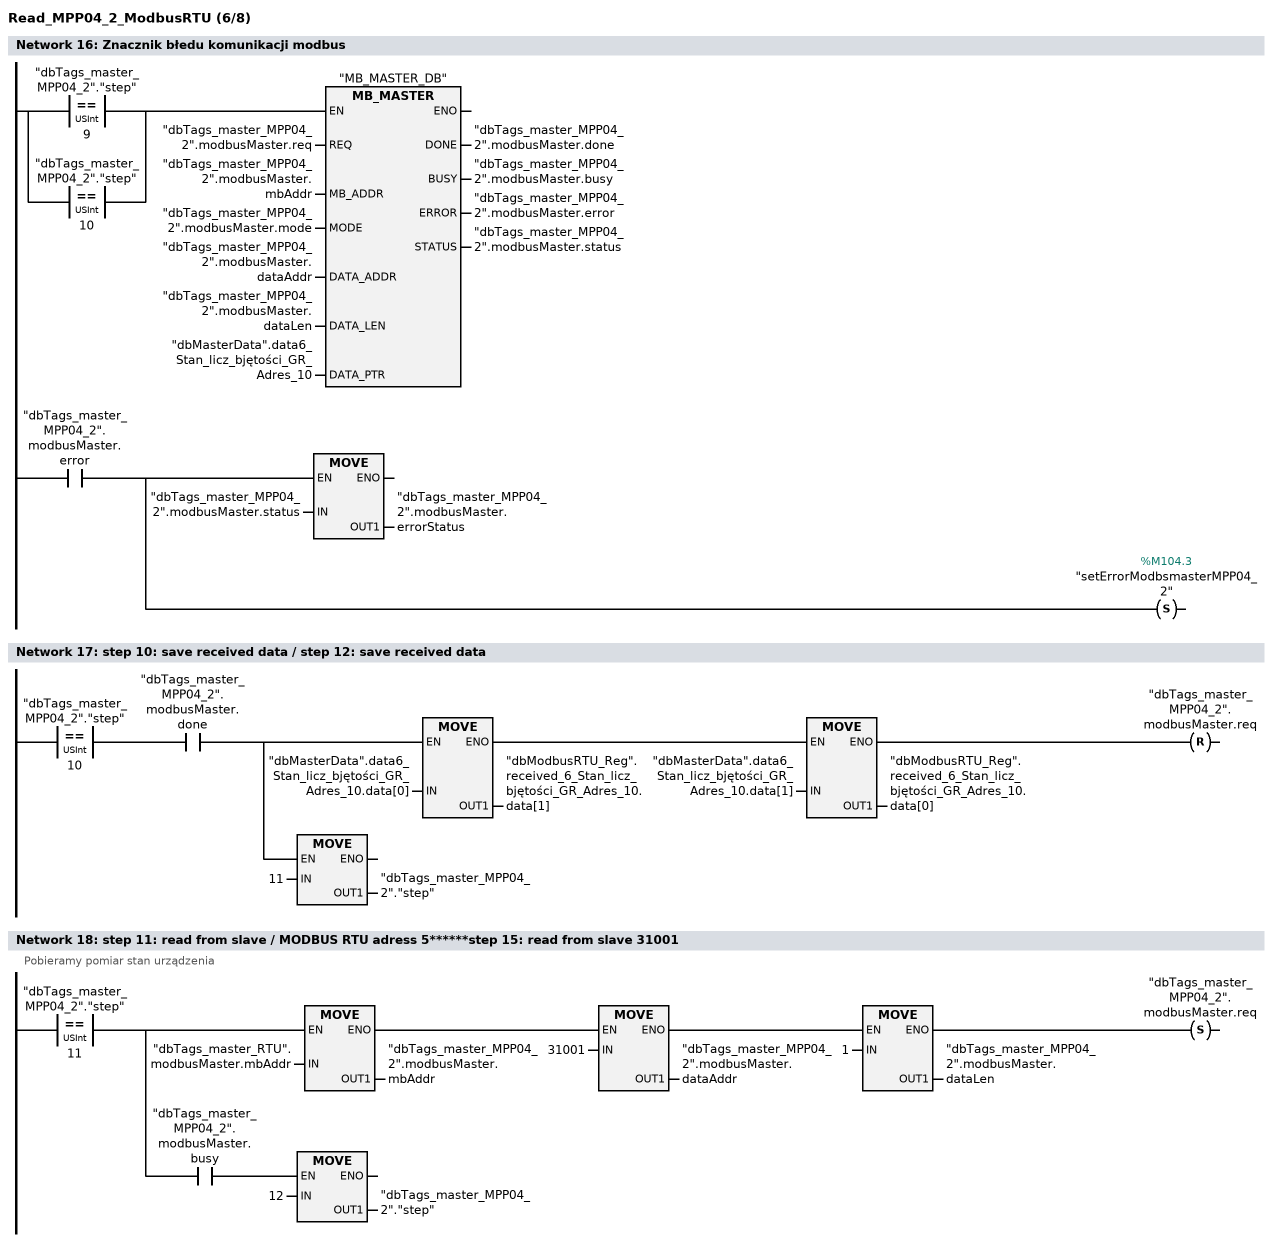
   RUNG wire#powerrail
      { S7_Templates := "SrcType := USInt" } EQ_Contact(in1 := "dbTags_master_MPP04_2"."step", in2 := 9)
      wire#w1
      "MB_MASTER_DB".MB_MASTER(REQ := "dbTags_master_MPP04_2".modbusMaster.req, MB_ADDR := "dbTags_master_MPP04_2".modbusMaster.mbAddr, MODE := "dbTags_master_MPP04_2".modbusMaster.mode, DATA_ADDR := "dbTags_master_MPP04_2".modbusMaster.dataAddr, DATA_LEN := "dbTags_master_MPP04_2".modbusMaster.dataLen, DATA_PTR := "dbMasterData".data6_Stan_licz_bjętości_GR_Adres_10, DONE => "dbTags_master_MPP04_2".modbusMaster.done, BUSY => "dbTags_master_MPP04_2".modbusMaster.busy, ERROR => "dbTags_master_MPP04_2".modbusMaster.error, STATUS => "dbTags_master_MPP04_2".modbusMaster.status)
   END_RUNG
   RUNG wire#powerrail
      { S7_Templates := "SrcType := USInt" } EQ_Contact(in1 := "dbTags_master_MPP04_2"."step", in2 := 10)
   END_RUNG wire#w1
   RUNG wire#powerrail
      Contact( "dbTags_master_MPP04_2".modbusMaster.error )
      wire#w2
      { S7_GenerateENO := "TRUE" } Move(in := "dbTags_master_MPP04_2".modbusMaster.status, out1 => "dbTags_master_MPP04_2".modbusMaster.errorStatus)
   END_RUNG
   RUNG wire#w2
      S_Coil( "setErrorModbsmasterMPP04_2" )
   END_RUNG
   // the same network as SCL:
   IF ("dbTags_master_MPP04_2"."step" = 9) OR ("dbTags_master_MPP04_2"."step" = 10) THEN
       "MB_MASTER_DB"(REQ := "dbTags_master_MPP04_2".modbusMaster.req,   // MB_MASTER
                      MB_ADDR := "dbTags_master_MPP04_2".modbusMaster.mbAddr,
                      MODE := "dbTags_master_MPP04_2".modbusMaster.mode,
                      DATA_ADDR := "dbTags_master_MPP04_2".modbusMaster.dataAddr,
                      DATA_LEN := "dbTags_master_MPP04_2".modbusMaster.dataLen,
                      DATA_PTR := "dbMasterData".data6_Stan_licz_bjętości_GR_Adres_10,
                      DONE => "dbTags_master_MPP04_2".modbusMaster.done,
                      BUSY => "dbTags_master_MPP04_2".modbusMaster.busy,
                      ERROR => "dbTags_master_MPP04_2".modbusMaster.error,
                      STATUS => "dbTags_master_MPP04_2".modbusMaster.status);
   END_IF;
   IF "dbTags_master_MPP04_2".modbusMaster.error THEN
       "dbTags_master_MPP04_2".modbusMaster.errorStatus := "dbTags_master_MPP04_2".modbusMaster.status;
       "setErrorModbsmasterMPP04_2" := TRUE;
   END_IF;
END_REGION

REGION Network 17: step 10: save received data / step 12: save received data
   RUNG wire#powerrail
      { S7_Templates := "SrcType := USInt" } EQ_Contact(in1 := "dbTags_master_MPP04_2"."step", in2 := 10)
      Contact( "dbTags_master_MPP04_2".modbusMaster.done )
      wire#w1
      { S7_GenerateENO := "TRUE" } Move(in := "dbMasterData".data6_Stan_licz_bjętości_GR_Adres_10.data[0], out1 => "dbModbusRTU_Reg".received_6_Stan_licz_bjętości_GR_Adres_10.data[1])
      { S7_GenerateENO := "TRUE" } Move(in := "dbMasterData".data6_Stan_licz_bjętości_GR_Adres_10.data[1], out1 => "dbModbusRTU_Reg".received_6_Stan_licz_bjętości_GR_Adres_10.data[0])
      R_Coil( "dbTags_master_MPP04_2".modbusMaster.req )
   END_RUNG
   RUNG wire#w1
      { S7_GenerateENO := "TRUE" } Move(in := 11, out1 => "dbTags_master_MPP04_2"."step")
   END_RUNG
   // the same network as SCL:
   // ENO of a box is taken as its EN; it also drops when the box reports an error
   IF ("dbTags_master_MPP04_2"."step" = 10) AND "dbTags_master_MPP04_2".modbusMaster.done THEN
       "dbModbusRTU_Reg".received_6_Stan_licz_bjętości_GR_Adres_10.data[1] := "dbMasterData".data6_Stan_licz_bjętości_GR_Adres_10.data[0];
       "dbModbusRTU_Reg".received_6_Stan_licz_bjętości_GR_Adres_10.data[0] := "dbMasterData".data6_Stan_licz_bjętości_GR_Adres_10.data[1];
       "dbTags_master_MPP04_2".modbusMaster.req := FALSE;
       "dbTags_master_MPP04_2"."step" := 11;
   END_IF;
END_REGION

REGION Network 18: step 11: read from slave / MODBUS RTU adress 5******step 15: read from slave 31001
   // Pobieramy pomiar stan urządzenia
   RUNG wire#powerrail
      { S7_Templates := "SrcType := USInt" } EQ_Contact(in1 := "dbTags_master_MPP04_2"."step", in2 := 11)
      wire#w1
      Move(in := "dbTags_master_RTU".modbusMaster.mbAddr, out1 => "dbTags_master_MPP04_2".modbusMaster.mbAddr)
      { S7_GenerateENO := "TRUE" } Move(in := 31001, out1 => "dbTags_master_MPP04_2".modbusMaster.dataAddr)
      Move(in := 1, out1 => "dbTags_master_MPP04_2".modbusMaster.dataLen)
      S_Coil( "dbTags_master_MPP04_2".modbusMaster.req )
   END_RUNG
   RUNG wire#w1
      Contact( "dbTags_master_MPP04_2".modbusMaster.busy )
      { S7_GenerateENO := "TRUE" } Move(in := 12, out1 => "dbTags_master_MPP04_2"."step")
   END_RUNG
   // the same network as SCL:
   // ENO of a box is taken as its EN; it also drops when the box reports an error
   #_w1 := "dbTags_master_MPP04_2"."step" = 11;
   IF #_w1 THEN
       "dbTags_master_MPP04_2".modbusMaster.mbAddr := "dbTags_master_RTU".modbusMaster.mbAddr;
       "dbTags_master_MPP04_2".modbusMaster.dataAddr := 31001;
       "dbTags_master_MPP04_2".modbusMaster.dataLen := 1;
       "dbTags_master_MPP04_2".modbusMaster.req := TRUE;
   END_IF;
   IF #_w1 AND "dbTags_master_MPP04_2".modbusMaster.busy THEN "dbTags_master_MPP04_2"."step" := 12; END_IF;
END_REGION

REGION Network 19: Znacznik błedu komunikacji modbus
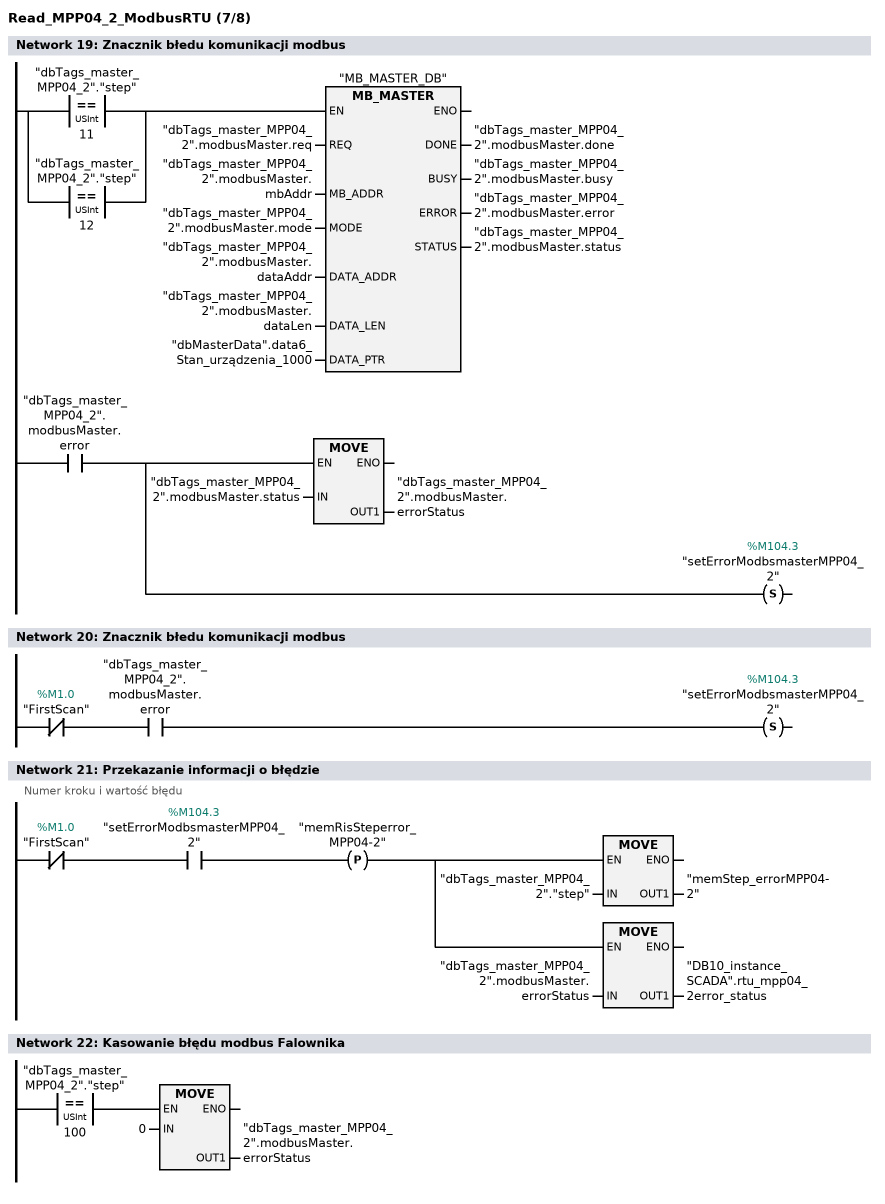
   RUNG wire#powerrail
      { S7_Templates := "SrcType := USInt" } EQ_Contact(in1 := "dbTags_master_MPP04_2"."step", in2 := 11)
      wire#w1
      "MB_MASTER_DB".MB_MASTER(REQ := "dbTags_master_MPP04_2".modbusMaster.req, MB_ADDR := "dbTags_master_MPP04_2".modbusMaster.mbAddr, MODE := "dbTags_master_MPP04_2".modbusMaster.mode, DATA_ADDR := "dbTags_master_MPP04_2".modbusMaster.dataAddr, DATA_LEN := "dbTags_master_MPP04_2".modbusMaster.dataLen, DATA_PTR := "dbMasterData".data6_Stan_urządzenia_1000, DONE => "dbTags_master_MPP04_2".modbusMaster.done, BUSY => "dbTags_master_MPP04_2".modbusMaster.busy, ERROR => "dbTags_master_MPP04_2".modbusMaster.error, STATUS => "dbTags_master_MPP04_2".modbusMaster.status)
   END_RUNG
   RUNG wire#powerrail
      { S7_Templates := "SrcType := USInt" } EQ_Contact(in1 := "dbTags_master_MPP04_2"."step", in2 := 12)
   END_RUNG wire#w1
   RUNG wire#powerrail
      Contact( "dbTags_master_MPP04_2".modbusMaster.error )
      wire#w2
      { S7_GenerateENO := "TRUE" } Move(in := "dbTags_master_MPP04_2".modbusMaster.status, out1 => "dbTags_master_MPP04_2".modbusMaster.errorStatus)
   END_RUNG
   RUNG wire#w2
      S_Coil( "setErrorModbsmasterMPP04_2" )
   END_RUNG
   // the same network as SCL:
   IF ("dbTags_master_MPP04_2"."step" = 11) OR ("dbTags_master_MPP04_2"."step" = 12) THEN
       "MB_MASTER_DB"(REQ := "dbTags_master_MPP04_2".modbusMaster.req,   // MB_MASTER
                      MB_ADDR := "dbTags_master_MPP04_2".modbusMaster.mbAddr,
                      MODE := "dbTags_master_MPP04_2".modbusMaster.mode,
                      DATA_ADDR := "dbTags_master_MPP04_2".modbusMaster.dataAddr,
                      DATA_LEN := "dbTags_master_MPP04_2".modbusMaster.dataLen,
                      DATA_PTR := "dbMasterData".data6_Stan_urządzenia_1000,
                      DONE => "dbTags_master_MPP04_2".modbusMaster.done,
                      BUSY => "dbTags_master_MPP04_2".modbusMaster.busy,
                      ERROR => "dbTags_master_MPP04_2".modbusMaster.error,
                      STATUS => "dbTags_master_MPP04_2".modbusMaster.status);
   END_IF;
   IF "dbTags_master_MPP04_2".modbusMaster.error THEN
       "dbTags_master_MPP04_2".modbusMaster.errorStatus := "dbTags_master_MPP04_2".modbusMaster.status;
       "setErrorModbsmasterMPP04_2" := TRUE;
   END_IF;
END_REGION

REGION Network 20: Znacznik błedu komunikacji modbus
   RUNG wire#powerrail
      I_Contact( "FirstScan" )
      Contact( "dbTags_master_MPP04_2".modbusMaster.error )
      S_Coil( "setErrorModbsmasterMPP04_2" )
   END_RUNG
   // the same network as SCL:
   IF NOT "FirstScan" AND "dbTags_master_MPP04_2".modbusMaster.error THEN
       "setErrorModbsmasterMPP04_2" := TRUE;
   END_IF;
END_REGION

REGION Network 21: Przekazanie informacji o błędzie
   // Numer kroku i wartość błędu
   RUNG wire#powerrail
      I_Contact( "FirstScan" )
      Contact( "setErrorModbsmasterMPP04_2" )
      P_Trig( "memRisSteperror_MPP04-2" )
      wire#w1
      Move(in := "dbTags_master_MPP04_2"."step", out1 => "memStep_errorMPP04-2")
   END_RUNG
   RUNG wire#w1
      { S7_GenerateENO := "TRUE" } Move(in := "dbTags_master_MPP04_2".modbusMaster.errorStatus, out1 => "DB10_instance_SCADA".rtu_mpp04_2error_status)
   END_RUNG
   // the same network as SCL:
   #_w1 := NOT "FirstScan" AND "setErrorModbsmasterMPP04_2";
   #_w2 := #_w1 AND NOT "memRisSteperror_MPP04-2";   // rising edge
   "memRisSteperror_MPP04-2" := #_w1;
   IF #_w2 THEN
       "memStep_errorMPP04-2" := "dbTags_master_MPP04_2"."step";
       "DB10_instance_SCADA".rtu_mpp04_2error_status := "dbTags_master_MPP04_2".modbusMaster.errorStatus;
   END_IF;
END_REGION

REGION Network 22: Kasowanie błędu modbus Falownika
   RUNG wire#powerrail
      { S7_Templates := "SrcType := USInt" } EQ_Contact(in1 := "dbTags_master_MPP04_2"."step", in2 := 100)
      { S7_GenerateENO := "TRUE" } Move(in := 0, out1 => "dbTags_master_MPP04_2".modbusMaster.errorStatus)
   END_RUNG
   // the same network as SCL:
   IF "dbTags_master_MPP04_2"."step" = 100 THEN
       "dbTags_master_MPP04_2".modbusMaster.errorStatus := 0;
   END_IF;
END_REGION

REGION Network 23: The enable to initiate a Modbus master request / step 16: save received data
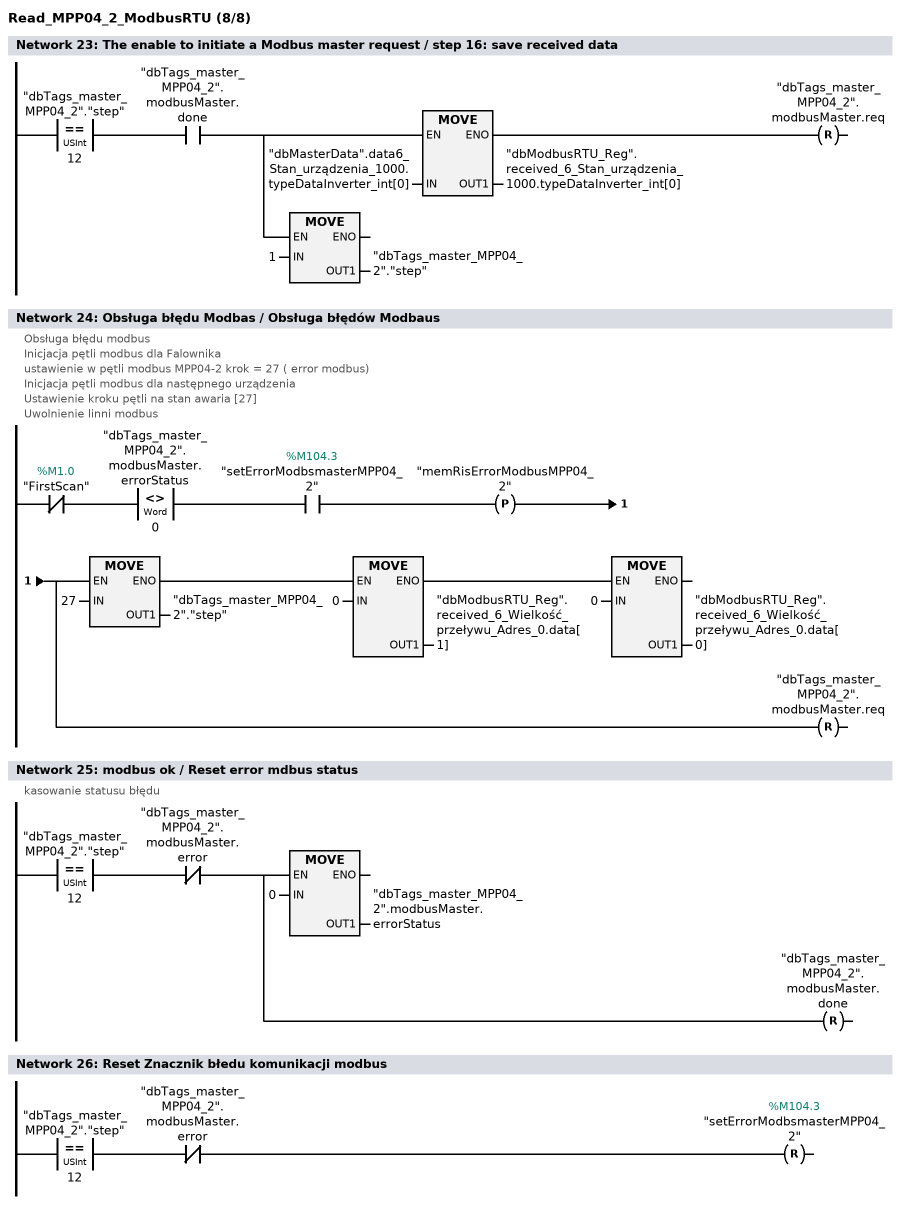
   RUNG wire#powerrail
      { S7_Templates := "SrcType := USInt" } EQ_Contact(in1 := "dbTags_master_MPP04_2"."step", in2 := 12)
      Contact( "dbTags_master_MPP04_2".modbusMaster.done )
      wire#w1
      { S7_GenerateENO := "TRUE" } Move(in := "dbMasterData".data6_Stan_urządzenia_1000.typeDataInverter_int[0], out1 => "dbModbusRTU_Reg".received_6_Stan_urządzenia_1000.typeDataInverter_int[0])
      R_Coil( "dbTags_master_MPP04_2".modbusMaster.req )
   END_RUNG
   RUNG wire#w1
      { S7_GenerateENO := "TRUE" } Move(in := 1, out1 => "dbTags_master_MPP04_2"."step")
   END_RUNG
   // the same network as SCL:
   // ENO of a box is taken as its EN; it also drops when the box reports an error
   IF ("dbTags_master_MPP04_2"."step" = 12) AND "dbTags_master_MPP04_2".modbusMaster.done THEN
       "dbModbusRTU_Reg".received_6_Stan_urządzenia_1000.typeDataInverter_int[0] := "dbMasterData".data6_Stan_urządzenia_1000.typeDataInverter_int[0];
       "dbTags_master_MPP04_2".modbusMaster.req := FALSE;
       "dbTags_master_MPP04_2"."step" := 1;
   END_IF;
END_REGION

REGION Network 24: Obsługa błędu Modbas / Obsługa błędów Modbaus
   // Obsługa błędu modbus 
   // Inicjacja pętli modbus dla Falownika
   // ustawienie w pętli modbus MPP04-2 krok = 27 ( error modbus)
   // Inicjacja pętli modbus dla następnego urządzenia
   // Ustawienie kroku pętli na stan awaria [27]
   // Uwolnienie linni modbus
   RUNG wire#powerrail
      I_Contact( "FirstScan" )
      { S7_Templates := "SrcType := Word" } NE_Contact(in1 := "dbTags_master_MPP04_2".modbusMaster.errorStatus, in2 := 0)
      Contact( "setErrorModbsmasterMPP04_2" )
      P_Trig( "memRisErrorModbusMPP04_2" )
      wire#w1
      { S7_GenerateENO := "TRUE" } Move(in := 27, out1 => "dbTags_master_MPP04_2"."step")
      { S7_GenerateENO := "TRUE" } Move(in := 0, out1 => "dbModbusRTU_Reg".received_6_Wielkość_przeływu_Adres_0.data[1])
      { S7_GenerateENO := "TRUE" } Move(in := 0, out1 => "dbModbusRTU_Reg".received_6_Wielkość_przeływu_Adres_0.data[0])
   END_RUNG
   RUNG wire#w1
      R_Coil( "dbTags_master_MPP04_2".modbusMaster.req )
   END_RUNG
   // the same network as SCL:
   // ENO of a box is taken as its EN; it also drops when the box reports an error
   #_w1 := NOT "FirstScan" AND ("dbTags_master_MPP04_2".modbusMaster.errorStatus <> 0) AND "setErrorModbsmasterMPP04_2";
   #_w2 := #_w1 AND NOT "memRisErrorModbusMPP04_2";   // rising edge
   "memRisErrorModbusMPP04_2" := #_w1;
   IF #_w2 THEN
       "dbTags_master_MPP04_2"."step" := 27;
       "dbModbusRTU_Reg".received_6_Wielkość_przeływu_Adres_0.data[1] := 0;
       "dbModbusRTU_Reg".received_6_Wielkość_przeływu_Adres_0.data[0] := 0;
       "dbTags_master_MPP04_2".modbusMaster.req := FALSE;
   END_IF;
END_REGION

REGION Network 25: modbus ok / Reset error mdbus status
   // kasowanie statusu błędu
   RUNG wire#powerrail
      { S7_Templates := "SrcType := USInt" } EQ_Contact(in1 := "dbTags_master_MPP04_2"."step", in2 := 12)
      I_Contact( "dbTags_master_MPP04_2".modbusMaster.error )
      wire#w1
      { S7_GenerateENO := "TRUE" } Move(in := 0, out1 => "dbTags_master_MPP04_2".modbusMaster.errorStatus)
   END_RUNG
   RUNG wire#w1
      R_Coil( "dbTags_master_MPP04_2".modbusMaster.done )
   END_RUNG
   // the same network as SCL:
   IF ("dbTags_master_MPP04_2"."step" = 12) AND NOT "dbTags_master_MPP04_2".modbusMaster.error THEN
       "dbTags_master_MPP04_2".modbusMaster.errorStatus := 0;
       "dbTags_master_MPP04_2".modbusMaster.done := FALSE;
   END_IF;
END_REGION

REGION Network 26: Reset Znacznik błedu komunikacji modbus
   RUNG wire#powerrail
      { S7_Templates := "SrcType := USInt" } EQ_Contact(in1 := "dbTags_master_MPP04_2"."step", in2 := 12)
      I_Contact( "dbTags_master_MPP04_2".modbusMaster.error )
      R_Coil( "setErrorModbsmasterMPP04_2" )
   END_RUNG
   // the same network as SCL:
   IF ("dbTags_master_MPP04_2"."step" = 12) AND NOT "dbTags_master_MPP04_2".modbusMaster.error THEN
       "setErrorModbsmasterMPP04_2" := FALSE;
   END_IF;
END_REGION
END_FUNCTION

FUNCTION "Zapis_Analogi_do_dbHold_ModbusTCP" : Void
TITLE = Przekazanie wartości 
{ S7_Optimized_Access := 'TRUE' }
AUTHOR : rtecmer
VERSION : 0.1
//Funkcja kopiuje wartości analogowe z db SCADA do db ModbusTCP 

BEGIN
	(*
	//=============================================================================
	//(JZWiK S.A Radosław Tecmer)
	//(c)Copyright (2022) All Rights Reserved
	//-----------------------------------------------------------------------------
	//Testowane z:   (system docelowy z  FW 4.4)
	//Pakiet inżynierski:   TIA Portal (V16 Update 5)
	//Ograniczenia:  ( - )
	//Wymagania:  (minimalne S7-1200 CPU 1215C FW 4.2 .)
	//Funkcjonalnośc: (Przekazanire aktualnego wartości pomiarów analogowych
	                    do dbHold modbusTCP )
	//-----------------------------------------------------------------------------
	//Zmainy wprowadzone:
	//Wersja  Data       Osoba wprowadzająca zmiany - ekspert
	//01.00.00 09.03.2022 (Tecmer Radosław - twórca) Pieresza wersja 01.00.00
	//=============================================================================
	*)
	
	// Analogi 
	
	REGION Analogi
	  // 
	  "dbHold_Sending".data.actB5_bar_magistrala :="DB10_instance_SCADA"."actCiśnienie-magistralaB5";
	  "dbHold_Sending".data.act_poziom_ZB1:="DB10_instance_SCADA".actPoziomZbiornik_1  ;
	  "dbHold_Sending".data.act_poziom_ZB2:= "DB10_instance_SCADA".actPoziomZbiornik_2  ;
	  "dbHold_Sending".data.act_poziom_ZB3:= "DB10_instance_SCADA".actPoziomZbiornik_3  ;
	  "dbHold_Sending".data.act_poziom_ZB4:=  "DB10_instance_SCADA".actPoziomZbiornik_4 ;
	  "dbHold_Sending".data.act_przepływ_VF_Q2:="DB10_instance_SCADA".actPrzepływ_Q2;
	 //dbHold_Sending".datat.act_przepływ-VR_Q2":=  ;
	  "dbHold_Sending".data.sum_przepływ_Q2:= "DB10_instance_SCADA".sumPrzepływVF_Q2 ;
	  "dbHold_Sending".data.stat.act_położenie_Z10 :="DB10_instance_SCADA".actPołożenieZ10 ;
	  
	END_REGION
	
	
END_FUNCTION

FUNCTION "Zapis_Status_Napedów_do_dbHold_ModbusTCP" : Void
TITLE = Przekazanie ststusu napedu
{ S7_Optimized_Access := 'TRUE' }
AUTHOR : rtecmer
VERSION : 0.1
//Funkcja przekazuje aktualny status napędu z bloku db SCADA do bloku db Hold Modbus TCP

BEGIN
	(*
	//=============================================================================
	//(JZWiK S.A Radosław Tecmer)
	//(c)Copyright (2022) All Rights Reserved
	//-----------------------------------------------------------------------------
	//Testowane z:   (system docelowy z  FW 4.4)
	//Pakiet inżynierski:   TIA Portal (V16 Update 5)
	//Ograniczenia:  ( - )
	//Wymagania:  (minimalne S7-1200 CPU 1215C FW 4.2 .)
	//Funkcjonalnośc: (Przekazanire aktualnego statusu napędu do bloku 
	                    danych dbHold modbusTCP )
	//-----------------------------------------------------------------------------
	//Zmainy wprowadzone:
	//Wersja  Data       Osoba wprowadzająca zmiany - ekspert
	//01.00.00 09.03.2022 (Tecmer Radosław - twórca) Pieresza wersja 01.00.00
	//=============================================================================
	*)
	
	REGION Zasuwy Status Napędu
	  // przeazanie
	  "dbHold_Sending".data.stat.status_Z1:="DB10_instance_SCADA".instZ1  ;
	  "dbHold_Sending".data.stat.status_Z2:= "DB10_instance_SCADA".instZ2 ;
	  "dbHold_Sending".data.stat.status_Z3:= "DB10_instance_SCADA".instZ3 ;
	  "dbHold_Sending".data.stat.status_Z4:= "DB10_instance_SCADA".instZ4 ;
	  "dbHold_Sending".data.stat.status_Z5:= "DB10_instance_SCADA".instZ5 ;
	  "dbHold_Sending".data.stat.status_Z6:= "DB10_instance_SCADA".instZ6 ;
	  "dbHold_Sending".data.stat.status_Z7:= "DB10_instance_SCADA".instZ7 ;
	  "dbHold_Sending".data.stat.status_Z8:= "DB10_instance_SCADA".instZ8 ;
	  "dbHold_Sending".data.stat.status_Z9:= "DB10_instance_SCADA".instZ9 ;
	  "dbHold_Sending".data.stat.status_Z10:= "DB10_instance_SCADA".instZ10 ;
	  
	END_REGION
	
END_FUNCTION

FUNCTION "Convertion_value_ModbusRTU" : Void
{ S7_Optimized_Access := 'TRUE' }
AUTHOR : rtecmer
VERSION : 0.1

BEGIN
	(*
	//=============================================================================
	//(JZWiK S.A Radosław Tecmer)
	//(c)Copyright (2021) All Rights Reserved
	//-----------------------------------------------------------------------------
	//Testowane z:   (system docelowy z  FW 4.2)
	//Pakiet inżynierski:   TIA Portal (V14 Sp1 Update 9)
	//Ograniczenia:  ( - )
	//Wymagania:  (minimalne S7-1200 CPU 1214 FW 3.2 .)
	//Funkcjonalnośc: (Przesuniecie bajtów (podobnie do funkcji SWAP) 
	//                  i przekazanie do bloku danych )
	//-----------------------------------------------------------------------------
	//Zmainy wprowadzone:
	//Wersja  Data       Osoba wprowadzająca zmiany - ekspert
	//01.00.00 31.01.2022 (Tecmer Radosław - twórca) Pieresza wersja 01.00.00
	//=============================================================================
	*)
	
	
	
	
	
	
	
	REGION Q2 przepływomierz
	  // Adres 0 - bierzący przepływ
	  "dbModbusRTU_Reg"."Przepływomierz nr2".received_6_przeływu_VF_Adres_0 := DWORD_TO_REAL(%DB37.DBD0);
	  
	  // warunek gdy komunikacja z przepływomierzem ok / błąd
	  IF "DB10_instance_SCADA".rtu_mpp04_2error_status = 0  THEN
	    // przepisz wartość z modbus rtu act przepływ 
	    "dbdane".Wielkość_przeływu_Q2 := "dbModbusRTU_Reg"."Przepływomierz nr2".received_6_przeływu_VF_Adres_0;
	  ELSE
	    "dbdane".Wielkość_przeływu_Q2 := 0.0;
	    ;
	  END_IF;
	  
	  
	  // Adres 2 - Licznik_objętość_VF
	  "dbModbusRTU_Reg"."Przepływomierz nr2".received_6_objętość_VF_Adres_2 := DWORD_TO_REAL(%DB37.DBD4);
	  
	  "dbdane".Licznik_objętość_VF_Q2 := "dbModbusRTU_Reg"."Przepływomierz nr2".received_6_objętość_VF_Adres_2;
	  
	  // Adres 4- stan bierzący licznika objetości w stecz VR
	  "dbModbusRTU_Reg"."Przepływomierz nr2"."received_6_objętośc RF_Adres_4" := DWORD_TO_REAL(%DB37.DBD8);
	  
	  "dbdane".Licznik_objętość_VR_Q2 := "dbModbusRTU_Reg"."Przepływomierz nr2"."received_6_objętośc RF_Adres_4";
	  
	  // Adres 6- stan bierzący licznika różnicowego  objętości VD
	  
	  
	  
	  // Adres 8- główny liczni objetości w przód GF
	  "dbModbusRTU_Reg"."Przepływomierz nr2".received_6_licznik_objętości_GF_Adres_8 := DWORD_TO_REAL(%DB37.DBD16);
	  
	  "dbdane".Stan_licz_bjętości_GF_Q2 := "dbModbusRTU_Reg"."Przepływomierz nr2".received_6_licznik_objętości_GF_Adres_8;
	  
	  // Adres 10- główny liczni objetości w stecz GR
	  "dbModbusRTU_Reg"."Przepływomierz nr2".received_6_Licznik_objętości_GR_Adres_10 := DWORD_TO_REAL(%DB37.DBD20);
	  
	  "dbdane".Stan_licz_rózicowego_obj_GD_Q2 := "dbModbusRTU_Reg"."Przepływomierz nr2".received_6_Licznik_objętości_GR_Adres_10;
	  
	  //Adres 12- główny lróznicowy liczni objetościGD
	  
	  
	  
	  // Status MP04 Q2 - magistrala
	  "dbModbusRTU_Reg"."Przepływomierz nr2".received_6_status_przepływomierza_Adres_1000 := "dbModbusRTU_Reg".received_6_Stan_urządzenia_1000.typeDataInverter_int[0];
	  "dbdane"._Stan_urządzenia_Q2 := "dbModbusRTU_Reg".received_6_Stan_urządzenia_1000.typeDataInverter_int[0];
	  
	  
	  
	  
	  
	  
	END_REGION
	
END_FUNCTION

FUNCTION "ClearError_Modbus" : Void
{ S7_Optimized_Access := 'TRUE' }
AUTHOR : rtecmer
VERSION : 0.1

BEGIN
	
	(*
	//=============================================================================
	//(JZWiK S.A Radosław Tecmer)
	//(c)Copyright (2021) All Rights Reserved
	//-----------------------------------------------------------------------------
	//Testowane z:   (system docelowy z  FW 4.4)
	//Pakiet inżynierski:   TIA Portal (V14 Sp1 Update 9)
	//Ograniczenia:  ( - )
	//Wymagania:  (minimalne S7-1200 CPU 1215C FW 4.2 .)
	//Funkcjonalnośc: (Obsługa błedów na magistrali Modbus RTU, inicjacja pętli po konfliktach )
	//-----------------------------------------------------------------------------
	//Zmainy wprowadzone:
	//Wersja  Data       Osoba wprowadzająca zmiany - ekspert
	//01.00.00 17.11.2021 (Tecmer Radosław - twórca) Pieresza wersja 01.00.00
	//=============================================================================
	*)
	
	
	
	REGION MPP04-2 Modbau RTU
	  // Sprawdzanie czy 
	  IF "dbTags_master_MPP04_2".step = 27 THEN
	    // Statement section IF
	    "dbTags_master_MPP04_2".modbusMaster.error := FALSE;
	    "dbTags_master_MPP04_2".modbusMaster.busy := FALSE;
	    "dbTags_master_MPP04_2".modbusMaster.status := 0;
	    //  "dbTags_master_MPP04_2".modbusMaster.errorStatus := 0;
	    "setErrorModbsmasterMPP04_2" := FALSE;
	    "dbTags_master_MPP04_2".step := 1;
	    
	    ;
	  END_IF;
	  
	  
	END_REGION
	
	//Modbus RTU Error Code RESET
	REGION Modbus RTU Error Code
	  // Ustaw reset modbus rtu
	  IF "DB10_instance_SCADA".rtu_step_reset THEN
	    // Ustawienie domyślnych strtowych 
	    "dbTags_master_MPP04_2".step := 12;
	   //"dbTags_master_MPP04_2".step := 25;
	
	    "DB10_instance_SCADA".rtu_step_reset := 0;
	    ;
	  END_IF;
	  
	  
	END_REGION
	
	// Ustawienie Błędu Modbus RTU 
	REGION Set Fault Modbus RTU 
	  // Jeśli zmienna kodu błędu różna od 0 to ustaw znacznik w błędu Modbus w bloku danych SCADA
	  // i przekaż wartość błędów
	  IF %DB10.DBX68.4 = TRUE OR"comunication_alarm_modbus_rtu" THEN
	    // przekazanie bładu statusu 
	    "DB10_instance_SCADA".rtu_mpp04_2error_status := "dbTags_master_MPP04_2".modbusMaster.errorStatus;
	 ELSE
	    ;
	    ;
	  END_IF;
	  
	  
	  // Modbus przekaż bit do instancji SCADA Alarm ostrzeżenie usterka z Modbau RTU
	  // Przynajmniej jeden slave nie odpowiada
	  IF 
	    "dbTags_master_MPP04_2".step = 27
	  THEN
	    %DB10.DBX68.4 := TRUE;
	
	    ;
	  ELSE
	    %DB10.DBX68.4 := FALSE;
	    
	  END_IF;
	  
	  
	  
	  
	  
	  
	END_REGION
	
	
	
	
	
END_FUNCTION

FUNCTION "Zatrzask Parametrów" : Void
TITLE = Kopiowanie do blkoków instancji 
{ S7_Optimized_Access := 'TRUE' }
AUTHOR : rtecmer
VERSION : 0.1
//Funkcja inicjowana znacznikiem ustawianym przez HMI po wprowadzeniu zmian, kopiuje dane z DB10 (SCADA) do instancji parametryzującej cały proces sterowania.

BEGIN
	(*
	//=============================================================================
	//(JZWiK S.A Radosław Tecmer)
	//(c)Copyright (2022) All Rights Reserved
	//-----------------------------------------------------------------------------
	//Testowane z:   (system docelowy z  FW 4.4)
	//Pakiet inżynierski:   TIA Portal (V16 Update 5)
	//Ograniczenia:  ( - )
	//Wymagania:  (minimalne S7-1200 CPU 1215C FW 4.2 .)
	//Funkcjonalnośc: (Cykliczne pobieranie danych konfiguracyjnych na potrzeby inicjacji danych
	                    konfiguracji po awarii, restarcie)
	//-----------------------------------------------------------------------------
	//Zmainy wprowadzone:
	//Wersja  Data       Osoba wprowadzająca zmiany - ekspert
	//01.00.00 09.03.2022 (Tecmer Radosław - twórca) Pieresza wersja 01.00.00
	//=============================================================================
	*)
	
	
	
	REGION Kopiowanie z DB10 SCADA
	  // pobierz dane
	  IF "FirstScan" = FALSE THEN
	    "Parametryzacja"."Setting Controll".ModelSterowania := "DB10_instance_SCADA".ModelSterowania;
	    "Parametryzacja"."Setting Controll".TrybSterowania := "DB10_instance_SCADA".TrybSterowania;
	    "Parametryzacja"."Setting Controll".setPoziomNapełniania := "DB10_instance_SCADA".setPoziomNapełniania;
	    "Parametryzacja"."Setting Controll".setPoziomOpróżnianai := "DB10_instance_SCADA".setPoziomOpróżnianai;
	    "Parametryzacja"."Status drivers".instZ1 := "DB10_instance_SCADA".instZ1;
	    "Parametryzacja"."Status drivers".instZ2 := "DB10_instance_SCADA".instZ2;
	    "Parametryzacja"."Status drivers".instZ3 := "DB10_instance_SCADA".instZ3;
	    "Parametryzacja"."Status drivers".instZ4 := "DB10_instance_SCADA".instZ4;
	    "Parametryzacja"."Status drivers".instZ5 := "DB10_instance_SCADA".instZ5;
	    "Parametryzacja"."Status drivers".instZ6 := "DB10_instance_SCADA".instZ6;
	    "Parametryzacja"."Status drivers".instZ7 := "DB10_instance_SCADA".instZ7;
	    "Parametryzacja"."Status drivers".instZ8 := "DB10_instance_SCADA".instZ8;
	    "Parametryzacja"."Status drivers".instZ9 := "DB10_instance_SCADA".instZ9;
	    "Parametryzacja"."Status drivers".instZ10 := "DB10_instance_SCADA".instZ10;
	    
	    // Czasy sterowania zasuwami 
	    "Parametryzacja"."Time Tanks".Start_napełnianie:= "DB10_instance_SCADA".actDTL_FillingOn ;
	    "Parametryzacja"."Time Tanks".Stop_napełnianie:= "DB10_instance_SCADA".actDTL_FillingOff ;
	    "Parametryzacja"."Time Tanks".Start_przetłaczanie_1:=  "DB10_instance_SCADA".actDTL_pumpingOn ;
	    "Parametryzacja"."Time Tanks".Stop_przetłaczanie_1:= "DB10_instance_SCADA".actDTL_pumpingOff ;
	    "Parametryzacja"."Time Tanks".Start_dosilanie_1:= "DB10_instance_SCADA".actDTL_RechargingOn ;
	    "Parametryzacja"."Time Tanks".Stop_dosilanie_1:= "DB10_instance_SCADA".actDTL_RechargingOff ;
	    
	    "ProcessMemory_Static_1_setChanging" := FALSE;
	    ;
	  END_IF;
	  
	  
	  
	END_REGION
	
	// Zasuwa Z10
	REGION pobranie nowej wartości położenia Z10
	  // Pobieraj nową wartośc tylko  gdy jest większa od '0' -
	  // '0' stan zamknięcia
	  IF "FirstScan" = FALSE AND "DB10_instance_SCADA".setPołożenieZ10 >= 2  THEN
	    // Statement section IF
	    "Parametryzacja"."Setting Controll".setPołożenieZ10 := "DB10_instance_SCADA".setPołożenieZ10;
	    ;
	  END_IF;
	  
	 
	  
	END_REGION
	
	REGION Zbiorniki
	  // bit blokowania zbiornika
	
	 
	  
	END_REGION
	
END_FUNCTION

FUNCTION "Kasowanie alarów" : Void   // FC9, LAD
{ S7_Optimized_Access := 'TRUE' }
AUTHOR : rtecmer
VERSION : 0.1
// (*
// //=============================================================================
// //(JZWiK S.A Radosław Tecmer)
// //(c)Copyright (2022) All Rights Reserved
// //-----------------------------------------------------------------------------
// //Testowane z:   (system docelowy z  FW 4.4)
// //Pakiet inżynierski:   TIA Portal (V16 Update 5)
// //Ograniczenia:  ( - )
// //Wymagania:  (minimalne S7-1200 CPU 1215C FW 4.2 .)
// //Funkcjonalnośc: (Kasowanie alarmów napedów przez HMI )
// //-----------------------------------------------------------------------------
// //Zmainy wprowadzone:
// //Wersja  Data       Osoba wprowadzająca zmiany - ekspert
// //01.00.00 09.03.2022 (Tecmer Radosław - twórca) Pieresza wersja 01.00.00
// //=============================================================================
// *)
// stored: AutoNumber true, IsIECCheckEnabled false, SetENOAutomatically false, UDAEnableTagReadback false
BEGIN

REGION Network 2 (SCL): Kasowanie alarmu Z10
   IF  "dbtags_Sterowanie".HMI.resetScreen_1 = TRUE THEN
     // Statement section IF
     IF "Hbit_Alarm_Z10" THEN
       // ustaw reset bit 
        %DB10. := TRUE;
       ;
     END_IF;
     IF "Hbit_Alarm_Z9" THEN
       // ustaw reset bit 
       %DB10. := TRUE;
       ;
     END_IF;

     // kasowanie momentu
     "setAlarm_Moment_Z_9" := FALSE;
     "setAlarm_Moment_Z_10" := FALSE;

     %DB10. := FALSE;
     %DB10. := FALSE;


     ;
   END_IF;

   //IF %DB10.DBX24.0 = FALSE THEN
     // Statement section IF
    // "dbtags_Sterowanie".HMI.resetScreen_1 := False;
   //  %DB10.DBX25.6 := FALSE;

   //  ;
   //END_IF;
END_REGION

REGION Network 3 (SCL): Kasowanie alarmu Z1 Z2
   IF "dbtags_Sterowanie".HMI.resetScreen_5 = TRUE THEN
     // Statement section IF
     IF "Hbit_Alarm_Z1" THEN
       // ustaw reset bit 
       %DB10. := TRUE;
       ;
     END_IF;
     IF "Hbit_Alarm_Z2" THEN
       // ustaw reset bit 
       %DB10. := TRUE;
       ;
     END_IF;


    // kasowanie momentu
     "setAlarm_Moment_Z_1" := FALSE;
     "setAlarm_Moment_Z_2" := FALSE;

     %DB10. := FALSE;
     %DB10. := FALSE;
     ;
   END_IF;
END_REGION

REGION Network 4 (SCL): Kasowanie alarmu Z3 Z4
   IF "dbtags_Sterowanie".HMI.resetScreen_4 = TRUE THEN
     // Statement section IF
     IF "Hbit_Alarm_Z3" THEN
       // ustaw reset bit 
       %DB10. := TRUE;
       ;
     END_IF;
     IF "Hbit_Alarm_Z4" THEN
       // ustaw reset bit 
       %DB10. := TRUE;
       ;
     END_IF;

     // kasowanie momentu
     "setAlarm_Moment_Z_3" := FALSE;
     "setAlarm_Moment_Z_4" := FALSE;

     %DB10. := FALSE;
     %DB10. := FALSE;
     ;
   END_IF;
END_REGION

REGION Network 5 (SCL): Kasowanie alarmu Z5 Z6
   IF "dbtags_Sterowanie".HMI.resetScreen_3 = TRUE THEN
     // Statement section IF
     IF "Hbit_Alarm_Z5" THEN
       // ustaw reset bit 
       %DB10. := TRUE;
       ;
     END_IF;
     IF "Hbit_Alarm_Z6" THEN
       // ustaw reset bit 
       %DB10. := TRUE;
       ;
     END_IF;

     // kasowanie momentu
     "setAlarm_Moment_Z_5" := FALSE;
     "setAlarm_Moment_Z_6" := FALSE;

     %DB10. := FALSE;
     %DB10. := FALSE;

     ;
   END_IF;
END_REGION

REGION Network 6 (SCL): Kasowanie alarmu Z7 Z8
   IF "dbtags_Sterowanie".HMI.resetScreen_2 = TRUE THEN
     // Statement section IF
     IF "Hbit_Alarm_Z7" THEN
       // ustaw reset bit 
       %DB10. := TRUE;
       ;
     END_IF;
     IF "Hbit_Alarm_Z8" THEN
       // ustaw reset bit 
       %DB10. := TRUE;
       ;
     END_IF;

     // kasowanie momentu
     "setAlarm_Moment_Z_7" := FALSE;
     "setAlarm_Moment_Z_8" := FALSE;

     %DB10. := FALSE;
     %DB10. := FALSE;

     ;
   END_IF;
END_REGION

REGION Network 11: Kasowanie alarmu Z1 Z2
END_REGION
END_FUNCTION

FUNCTION_BLOCK "Alarm_magistrala_B5"
TITLE = Alarm ciśnieia na magistrali czyjnik B5
{ S7_Optimized_Access := 'TRUE' }
AUTHOR : rtecmer
VERSION : 0.1
//Zarządzanie alarmami od ciśnienia na magistrali (B5) DN500
   VAR_OUTPUT 
      bit_alarm_magistrala_min { ExternalAccessible := 'False'; ExternalVisible := 'False'; ExternalWritable := 'False'} : Bool := false;   // bit alarmmagistrala awaria niskie ciśnienie
      setControl_alarm_B5 { ExternalAccessible := 'False'; ExternalVisible := 'False'; ExternalWritable := 'False'} : Bool;   // Załczenie sterowania zbiornikami w trybie awarii na magistrali
   END_VAR

   VAR_IN_OUT 
      bit_off_alarm_niskie_magistrala { ExternalAccessible := 'False'; ExternalVisible := 'False'; ExternalWritable := 'False'} : Bool;   // bit koniec alarmu niskie bar magistrala
   END_VAR

   VAR 
      bit_normalne_magistrala { ExternalAccessible := 'False'; ExternalVisible := 'False'; ExternalWritable := 'False'} : Bool;   // bit detekcjinormalnego cisnienia magistrala
      memTriger_Strategia { ExternalAccessible := 'False'; ExternalVisible := 'False'; ExternalWritable := 'False'} : Bool;
      bit_niskie_magistrala { ExternalAccessible := 'False'; ExternalVisible := 'False'; ExternalWritable := 'False'} : Bool;   // bit detekcji niskiego cisnienia magistrala
   END_VAR


BEGIN
	(*
	//=============================================================================
	//(JZWiK S.A Radosław Tecmer)
	//(c)Copyright (2021) All Rights Reserved
	//-----------------------------------------------------------------------------
	//Testowane z:   (system docelowy z  FW 4.4)
	//Pakiet inżynierski:   TIA Portal (V14 Sp1 Update 9)
	//Ograniczenia:  ( - )
	//Wymagania:  (minimalne S7-1200 CPU 1215C FW 4.2 .)
	//Funkcjonalnośc: (Kontrola stanu ciśnienia na magistrali DN500, B5. Kontrola
	                   poziomu w zbiornikach i zarządznie wrybem awaryjnym otwarcia 
	                   Z9, odpływów ze zbiorników i zamknięcia dolotu do zbiorników
	                                                   )
	//-----------------------------------------------------------------------------
	//Zmainy wprowadzone:
	//Wersja  Data       Osoba wprowadzająca zmiany - ekspert
	//01.00.00 17.11.2021 (Tecmer Radosław - twórca) Pieresza wersja 01.00.00
	//=============================================================================
	*)
	
	
	REGION Kontrola  ciśnieia magistrali, alarm niskie magistrala czujnik B5
	  
	  // Kontrola ciśnienia zasilania z magistrali B5
	  // Detekcja zaistnienia awarii zasilania na magistrali
	  IF "DB10_instance_SCADA"."actCiśnienie-magistralaB5" < "Parametryzacja"."Setting Controll".alarmMin_CiśnienieGranica THEN
	    // Ustaw bit za niskie ciśnienie
	    #bit_niskie_magistrala := TRUE;
	  ELSE
	    
	    ;
	  END_IF;
	  
	  
	  
	  // Sprawdzanie powrotu zasilania z magistrali czujnik B5
	  IF "DB10_instance_SCADA"."actCiśnienie-magistralaB5" > 7.4 THEN
	    // Ustaw bit normalne ciśnienie
	    #bit_normalne_magistrala := TRUE;
	    
	  ELSE
	    #bit_normalne_magistrala := FALSE;
	    ;
	  END_IF;
	  
	  //Histerez na powrót normalnego zasilania z magistrali
	   "IEC_Timer_reserAlarmNiskie_cisnienie_DB".TON(IN:=#bit_normalne_magistrala,
	                                                PT:=T#5M,
	                                                Q=>#bit_off_alarm_niskie_magistrala);
	  
	
	  IF #bit_off_alarm_niskie_magistrala THEN
	    // kasowanie alarm niskie magistrala
	    #bit_niskie_magistrala := FALSE;
	    ;
	  END_IF;
	  
	  
	  // Histereza na ustawienie alarmu "niskie ćiśnienie na magistrali"
	  "IEC_Timer_setAlarmNiskie_ciśnienie_DB".TON(IN := #bit_niskie_magistrala,
	                                              PT := T#14M,
	                                              Q => #bit_alarm_magistrala_min);
	  
	
	  
	END_REGION
	
	
	
	REGION Awaryjne uruchamianie sterowania zbiornikami
	  // jeśli alarm magistrali
	  IF  #bit_alarm_magistrala_min  THEN
	    // ustaw znacznik
	    #setControl_alarm_B5 := TRUE;
	    ;
	  END_IF;
	  
	  // Jeśli koniec alarmu i zamknieta Z9  
	  IF #bit_off_alarm_niskie_magistrala AND "Hbit_Zamknieta_Z9" THEN
	    // resetuj znacznik 
	    #setControl_alarm_B5 := FALSE;
	    ;
	  END_IF;
	  
	  
	  
	END_REGION
	
END_FUNCTION_BLOCK

FUNCTION "D_IN" : Void
TITLE = Przekazanie wartości
{ S7_Optimized_Access := 'TRUE' }
AUTHOR : rtecmer
VERSION : 0.1
//Mapownaie wejść cyfrowych

BEGIN
	(*
	//=============================================================================
	//(JZWiK S.A Radosław Tecmer)
	//(c)Copyright (2021) All Rights Reserved
	//-----------------------------------------------------------------------------
	//Testowane z:   (system docelowy z  FW 4.2)
	//Pakiet inżynierski:   TIA Portal (V14 Sp1 Update 9)
	//Ograniczenia:  ( - )
	//Wymagania:  (minimalne S7-1200 CPU 1214 FW 3.2 .)
	//Funkcjonalnośc: (Mapowanie wejść cyfrowych )
	//-----------------------------------------------------------------------------
	//Zmainy wprowadzone:
	//Wersja  Data       Osoba wprowadzająca zmiany - ekspert
	//01.00.00 28.01.2022 (Tecmer Radosław - twórca) Pieresza wersja 01.00.00
	//=============================================================================
	*)
	
	// Zbiorniki pływaki minimum
	REGION pływaki
	  // przekazanie stanu
	  "float_min_tank_1" := "I2.5";
	  "float_min_tank_2" := "I2.6";
	  "float_min_tank_3" := "I2.7";
	  "float_min_tank_4" := "I3.0";
	  "float_max_tank_1" := "I5.5";
	  "float_max_tank_2" := "I5.6";
	  "float_max_tank_3" := "I5.7";
	  "float_max_tank_4" := "I6.0";
	  
	  
	END_REGION
	
	
	
	// Zasuwy
	"inputREM_Zasuwy" := "I6.1";
	
	REGION ZASUWA Z1 
	  // przekazanie wartości wspólne z MODACT MOK250 i AUMA
	  
	  "inputREMT_Z_1" := "inputREM_Zasuwy";
	  "inputOtwartaZ_1" := "I0.5";
	  "inputZamkniętaZ_1" := "I0.6";
	  "inputRuch_Z_1" := "I0.3";
	 // 
	  //momentówki normalny stan 1 awaria 0
	  "inputAwariaMomentZ_1" := "I0.4";
	  
	  // przekazanie wartości z AUMA
	  "inputAumagotowośćZ_1" := "I6.4";
	  "inputAumaautomatZ_1" := "I6.3";
	  "inputAumalokalneZ_1" := "I6.2";
	  
	  
	END_REGION
	
	REGION ZASUWA Z2 
	  // przekazanie wartości wspólne z MODACT MOK250 i AUMA
	  
	  "inputREMT_Z_2" := "inputREM_Zasuwy";
	  "inputOtwartaZ_2" := "I3.7";
	  "inputZamkniętaZ_2" := "I4.0";
	  "inputRuch_Z_2" := "I3.5";
	  //momentówki normalny stan 1 awaria 0
	  "inputAwariaMomentZ_2" := "I3.6";
	  
	  // przekazanie wartości z AUMA
	  "inputAumagotowośćZ_2" := "I6.7";
	  "inputAumaautomatZ_2" := "I6.6";
	  "inputAumalokalneZ_2" := "I6.5";
	  
	  
	END_REGION
	
	REGION ZASUWA Z3 
	  // przekazanie wartości wspólne z MODACT MOK250 i AUMA
	  
	  "inputREMT_Z_3" := "inputREM_Zasuwy";
	  "inputOtwartaZ_3" := "I1.1";
	  "inputZamkniętaZ_3" := "I1.2";
	  "inputRuch_Z_3" := "I0.7";
	  //momentówki normalny stan 1 awaria 0
	  "inputAwariaMomentZ_3" := "I1.0";
	  
	  // przekazanie wartości z AUMA
	  "inputAumagotowośćZ_3" := "I7.2";
	  "inputAumaautomatZ_3" := "I7.1";
	  "inputAumalokalneZ_3" := "I7.0";
	  
	  
	END_REGION
	
	REGION ZASUWA Z4 
	  // przekazanie wartości wspólne z MODACT MOK250 i AUMA
	  
	  "inputREMT_Z_4" := "inputREM_Zasuwy";
	  "inputOtwartaZ_4" := "I4.3";
	  "inputZamkniętaZ_4" := "I4.4";
	  "inputRuch_Z_4" := "I4.1";
	  //momentówki normalny stan 1 awaria 0
	  "inputAwariaMomentZ_4" := "I4.2";
	  
	  // przekazanie wartości z AUMA
	  "inputAumagotowośćZ_4" := "I7.5";
	  "inputAumaautomatZ_4" := "I7.4";
	  "inputAumalokalneZ_4" := "I7.3";
	  
	  
	END_REGION
	
	REGION ZASUWA Z5 
	  // przekazanie wartości wspólne z MODACT MOK250 i AUMA
	  
	  "inputREMT_Z_5" := "inputREM_Zasuwy";
	  "inputOtwartaZ_5" := "I1.5";
	  "inputZamkniętaZ_5" := "I2.0";
	  "inputRuch_Z_5" := "I1.3";
	  //momentówki normalny stan 1 awaria 0
	  "inputAwariaMomentZ_5" := "I1.4";
	  
	  // przekazanie wartości z AUMA
	  "inputAumagotowośćZ_5" := "I8.0";
	  "inputAumaautomatZ_5" := "I7.7";
	  "inputAumalokalneZ_5" := "I7.6";
	  
	  
	END_REGION
	
	REGION ZASUWA Z6 
	  // przekazanie wartości wspólne z MODACT MOK250 i AUMA
	  
	  "inputREMT_Z_6" := "inputREM_Zasuwy";
	  "inputOtwartaZ_6" := "I4.7";
	  "inputZamkniętaZ_6" := "I5.0";
	  "inputRuch_Z_6" := "I4.5";
	  //momentówki normalny stan 1 awaria 0
	  "inputAwariaMomentZ_6" := "I4.6";
	  
	  // przekazanie wartości z AUMA
	  "inputAumagotowośćZ_6" := "I8.3";
	  "inputAumaautomatZ_6" := "I8.2";
	  "inputAumalokalneZ_6" := "I8.1";
	  
	  
	END_REGION
	
	REGION ZASUWA Z7 
	  // przekazanie wartości wspólne z MODACT MOK250 i AUMA
	  
	  "inputREMT_Z_7" := "inputREM_Zasuwy";
	  "inputOtwartaZ_7" := "I2.3";
	  "inputZamkniętaZ_7" := "I2.4";
	  "inputRuch_Z_7" := "I2.1";
	  //momentówki normalny stan 1 awaria 0
	  "inputAwariaMomentZ_7" := "I2.2";
	  
	  // przekazanie wartości z AUMA
	  "inputAumagotowośćZ_7" := "I8.6";
	  "inputAumaautomatZ_7" := "I8.5";
	  "inputAumalokalneZ_7" := "I8.4";
	  
	  
	END_REGION
	
	REGION ZASUWA Z8 
	  // przekazanie wartości wspólne z MODACT MOK250 i AUMA
	  
	  "inputREMT_Z_8" := "inputREM_Zasuwy";
	  "inputOtwartaZ_8" := "I5.3";
	  "inputZamkniętaZ_8" := "I5.4";
	  "inputRuch_Z_8" := "I5.1";
	  //momentówki normalny stan 1 awaria 0
	  "inputAwariaMomentZ_8" := "I5.2";
	  
	  // przekazanie wartości z AUMA
	  "inputAumagotowośćZ_8" := "I9.1";
	  "inputAumaautomatZ_8" := "I9.0";
	  "inputAumalokalneZ_8" := "I8.7";
	  
	  
	END_REGION
	
	REGION ZASUWA Z9
	  // przekazanie wartości wspólne z MODACT MOK250 i AUMA
	  
	  "inputREMT_Z_9" := "inputREM_Zasuwy";
	  "inputOtwartaZ_9" := "I0.2";
	  "inputZamkniętaZ_9" := "I10.0";
	  "inputRuch_Z_9" := "I0.0";
	  //momentówki normalny stan 1 awaria 0
	  "inputAwariaMomentZ_9" := "I0.1";
	  
	  // przekazanie wartości z AUMA
	  "inputAumagotowośćZ_9" := "I9.4";
	  "inputAumaautomatZ_9" := "I9.3";
	  "inputAumalokalneZ_9" := "I9.2";
	  
	  
	END_REGION
	
	
	REGION ZASUWA Z10 
	  // przekazanie wartości  AUMA
	  
	  "inputREMT_Z_10" := "inputREM_Zasuwy";
	  IF "I3.3" = TRUE OR ("DB10_instance_SCADA".actPołożenieZ10 >= 3) THEN
	    // też otwarta 
	    "inputOtwartaZ_10" := TRUE;
	  ELSE
	    "inputOtwartaZ_10" := FALSE;
	    ;
	  END_IF;
	  
	  "inputOtwartaZ_10" := "I3.3";
	  IF ("DB10_instance_SCADA".actPołożenieZ10 <= 1) OR  ("I3.4" = TRUE) THEN
	    // też zamknieta
	    "isClose_od_położenia" := TRUE;
	  ELSE
	    "isClose_od_położenia" := FALSE;
	    ;
	  END_IF;
	  
	  "inputZamkniętaZ_10" := "I3.4";
	  "inputRuch_Z_10" := "I3.1";
	  //Auma nie wystawia osobnego sygnału awaria momentu wszystko na gotowość
	  //"inputAwariaMomentZ_10" := ;
	  
	  // przekazanie wartości z AUMA
	  "inputAumagotowośćZ_10" := "I9.7";
	  "inputAumaautomatZ_10" := "I9.6";
	  "inputAumalokalneZ_10" := "I9.5";
	  
	  
	END_REGION
END_FUNCTION

FUNCTION "AI_IN" : Void
TITLE = Przekazanie wartości analogowej
{ S7_Optimized_Access := 'TRUE' }
AUTHOR : rtecmer
VERSION : 0.1
//Mapownie wejść analogowych

BEGIN
	(*
	//=============================================================================
	//(JZWiK S.A Radosław Tecmer)
	//(c)Copyright (2021) All Rights Reserved
	//-----------------------------------------------------------------------------
	//Testowane z:   (system docelowy z  FW 4.2)
	//Pakiet inżynierski:   TIA Portal (V14 Sp1 Update 9)
	//Ograniczenia:  ( - )
	//Wymagania:  (minimalne S7-1200 CPU 1214 FW 3.2 .)
	//Funkcjonalnośc: (Mapowanie wejść analogowych )
	//-----------------------------------------------------------------------------
	//Zmainy wprowadzone:
	//Wersja  Data       Osoba wprowadzająca zmiany - ekspert
	//01.00.00 28.01.2022 (Tecmer Radosław - twórca) Pieresza wersja 01.00.00
	//=============================================================================
	*)
	
	
	
	// odczyt bezpośredni z AI
	
	IF "IW78":P >= 0.0 THEN // czy nie uszkodzone rury
	  IF "IW78":P < 27651 THEN // przerwana pętla prądowa
	    // to przekazanie wartości
	    "AI_położenie_Z10" := "IW78":P;
	    ;
	  ELSE
	    "AI_położenie_Z10" := 32767;
	    ;
	  END_IF;
	  
	  ;
	END_IF;
	
	
	// odczyt analogów przez OB30
	(*
	IF "IW76":P > 0.2 THEN // czy nie uszkodzone rury
	  IF "IW76":P < 27651 THEN // przerwana pętla prądowa
	    // to przekazanie wartości
	    "AI_ciśnienie_B5" := "IW76":P;
	    ;
	  ELSE
	    "AI_ciśnienie_B5" := 32767;
	    ;
	  END_IF;
	  
	  ;
	END_IF;
	
	*)
	
	//Symulacja czujnika B5
	//"AI_ciśnienie_B5" := "Zmienne_sterujące_zbiorników".testowy1 ;
	
	
	// odczyt poprzez filtr KALMANA funkcja FB11
	
	"filtr _kalmana_1_DB"();
	
	
END_FUNCTION

FUNCTION "Błąd nadajnika położenia" : Void
TITLE = Detekcja błędu nadajnika
{ S7_Optimized_Access := 'TRUE' }
AUTHOR : rtecmer
VERSION : 0.1
//Funkcja w oparciu o sygnały z czujników krańcowych położenia prądu 4-20mA nadajnika ustala czy wystąpił błąd nadajnika
   VAR_INPUT 
      isOpen : Bool;   // sygnał potwierdzenia otwarcia
      isClose : Bool;   // sygnał potwierdzenia zamknięcia
      actPosition : Word;   // sygnał aktualnego położenie 4-20mA
   END_VAR

   VAR_OUTPUT 
      isError_Position : Bool;   // sygnalizacja błędu pozycji
   END_VAR


BEGIN
	(*
	//=============================================================================
	//(JZWiK S.A Radosław Tecmer)
	//(c)Copyright (2021) All Rights Reserved
	//-----------------------------------------------------------------------------
	//Testowane z:   (system docelowy z  FW 4.4)
	//Pakiet inżynierski:   TIA Portal (V14 Sp1 Update 9)
	//Ograniczenia:  ( - )
	//Wymagania:  (minimalne S7-1200 CPU 1215C FW 4.2 .)
	//Funkcjonalnośc: (Detekcja błędu nadajnika prądowego
	//                  w oparciu o czujniki krańcowe położenia )
	//-----------------------------------------------------------------------------
	//Zmainy wprowadzone:
	//Wersja  Data       Osoba wprowadzająca zmiany - ekspert
	//01.00.00 05.02.2022 (Tecmer Radosław - twórca) Pieresza wersja 01.00.00
	//=============================================================================
	*)
	
	REGION Bład na Otwarcie
	  // Jeśli sygnał z krańcówki otwarta =1
	  IF #isOpen THEN
	    IF (#actPosition >= 28538) OR (#actPosition < 27381)  THEN
	      // ustaw sygnał błędu
	      #isError_Position := TRUE;
	    END_IF;
	    
	    // koniec
	    ;
	  END_IF;
	  
	 
	  
	END_REGION
	
	REGION Bład na Zamknięcie
	  // Jeśli sygnał z krancówki zamknięta =1
	  IF #isClose THEN
	    IF (#actPosition > 268 AND #actPosition < 65529) THEN
	      // ustaw sygnał błedu
	      #isError_Position := TRUE;
	    END_IF;
	    
	    // koniec
	    ;
	  END_IF;
	  
	  
	  
	END_REGION
	
	
END_FUNCTION

FUNCTION_BLOCK "AI_Scalowani_Położenia_Z10"
TITLE = Detekcja błędu położenia
{ S7_Optimized_Access := 'TRUE' }
AUTHOR : rtecmer
VERSION : 0.1
//Przekazanie do skalowania wartości z zakresu 0-27648
   VAR_INPUT 
      actAI_położenie_Z10 { ExternalAccessible := 'False'; ExternalVisible := 'False'; ExternalWritable := 'False'} : Word;   // aktualny sygnał analogowy położenia Z10
   END_VAR

   VAR_OUTPUT 
      isPosition : Bool;   // bit zasuwa na pozycji
   END_VAR

   VAR_TEMP 
      tmpAI_położenie_Z10 : Word;   // pomocniczy sygnał analogowy położenia Z10
      tmpSetVectorZ10 : Int;   // zadane położenie
      tempActVector_Z10 : Int;   // odczytane położenie
   END_VAR


BEGIN
	(*
	//=============================================================================
	//(JZWiK S.A Radosław Tecmer)
	//(c)Copyright (2021) All Rights Reserved
	//-----------------------------------------------------------------------------
	//Testowane z:   (system docelowy z  FW 4.2)
	//Pakiet inżynierski:   TIA Portal (V14 Sp1 Update 9)
	//Ograniczenia:  ( - )
	//Wymagania:  (minimalne S7-1200 CPU 1214 FW 3.2 .)
	//Funkcjonalnośc: (Detekcja błędu i skalowanie wejść analogowych połóżenie Z10 )
	//-----------------------------------------------------------------------------
	//Zmainy wprowadzone:
	//Wersja  Data       Osoba wprowadzająca zmiany - ekspert
	//01.00.00 28.01.2022 (Tecmer Radosław - twórca) Pieresza wersja 01.00.00
	//=============================================================================
	*)
	
	REGION Detekcja przekroczenia zakresu analogowego nadajnika Z10
	  // Przekazanie wartości położenia wtedy gdy jest w skali 4-20mA
	  // Jeśli przewód odłączony lub sygnał poza zakresem wprzkazanie wartości '0' 
	  
	  // Wartość zawysoka
	  IF (#actAI_położenie_Z10 >= "analog_error_H") THEN
	    // Przekazanie wartości domyślnej 0
	    #tmpAI_położenie_Z10 := 0;
	    ;
	  END_IF;
	  // Wartość poprawna
	  IF (#actAI_położenie_Z10 <= "analog_error_H") AND (#actAI_położenie_Z10 >= 0) THEN
	    // przekazanie własciwego sygnału 
	    #tmpAI_położenie_Z10 := #actAI_położenie_Z10;
	    ;
	  END_IF;
	  
	  
	  
	END_REGION
	
	
	REGION Położenie zasuwy Z10
	  // Konwersja i skalowanie 
	  // Jesli bedzie konieczne do dostroić parametr x0 około 5600 ( wartość zera z nadajnika)
	  "dbtags_Sterowanie"."Z10 Pozycja".encoder := "SclScaleLinearInt"(x := #tmpAI_położenie_Z10,
	                                                               yMin := 0,
	                                                               yMax := 100,
	                                                               x0 := 0,
	                                                               y0 := 0,
	                                                               x1 := 27648,
	                                                               y1 := 100);
	  
	END_REGION
	
	// ustawienie bitu Z10 na pozycji na potrzeby HMI
	REGION _name_
	  // 
	  #tmpSetVectorZ10 := "DB10_instance_SCADA".setPołożenieZ10;
	  #tempActVector_Z10 := "DB10_instance_SCADA".actPołożenieZ10;
	  
	  IF #tempActVector_Z10 = #tmpSetVectorZ10 THEN
	    // ustaw znacznik zasuwa na pozycji
	    #isPosition := TRUE;
	  ELSE
	    #isPosition:= FALSE
	    ;
	  END_IF;
	  
	  
	  
	  
	END_REGION
	
	
	
	
END_FUNCTION_BLOCK

FUNCTION "AI_IN_Scalowanie" : Void
TITLE = Konwersja wartości procesowej 
{ S7_Optimized_Access := 'TRUE' }
AUTHOR : rtecmer
VERSION : 0.1
//Obsługa przetworników analogowych. Konwersja i skalowanie wartości procesowych. 

BEGIN
	(*
	//=============================================================================
	//(JZWiK S.A Radosław Tecmer)
	//(c)Copyright (2021) All Rights Reserved
	//-----------------------------------------------------------------------------
	//Testowane z:   (system docelowy z  FW 4.2)
	//Pakiet inżynierski:   TIA Portal (V14 Sp1 Update 9)
	//Ograniczenia:  ( - )
	//Wymagania:  (minimalne S7-1200 CPU 1214 FW 3.2 .)
	//Funkcjonalnośc: (Konwersja i skalowanie wejść analogowych )
	//-----------------------------------------------------------------------------
	//Zmainy wprowadzone:
	//Wersja  Data       Osoba wprowadzająca zmiany - ekspert
	//01.00.00 28.01.2022 (Tecmer Radosław - twórca) Pieresza wersja 01.00.00
	//=============================================================================
	*)
	
	// Odczyt analogów poprzez filtr Kolmana
	REGION Analogi filtr kolmana ciśnienie sieci B5 i zbiorniki Zb1 - 4 
	  // Konwersja i skalowanie pomiarów z wyjścia funkcji filtru Kolmana (FB11)
	  //zbiornik 1
	  IF "KALMAN_DB".kalman_napiecie[0] > 9.9 THEN
	    // błąd pomiaru (przerwa w obwodzie) ustaw 0
	    "dbtags_Sterowanie"."Analog pomiar".kolman_poziom_zbiornik_1 := 0.0;
	  ELSE
	    // pomiar ok
	    "dbtags_Sterowanie"."Analog pomiar".kolman_poziom_zbiornik_1 := (100 * "KALMAN_DB".kalman_napiecie[0]);
	    ;
	  END_IF;
	  // zbiornik 2
	  IF "KALMAN_DB".kalman_napiecie[1] > 9.9 THEN
	    // błąd pomiaru (przerwa w obwodzie) ustaw 0
	    "dbtags_Sterowanie"."Analog pomiar".kolman_poziom_zbiornik_2 := 0.0;
	  ELSE
	    // pomiar ok
	    "dbtags_Sterowanie"."Analog pomiar".kolman_poziom_zbiornik_2 := (100 * "KALMAN_DB".kalman_napiecie[1]);
	    ;
	  END_IF;
	  // zbiornik 3
	  IF "KALMAN_DB".kalman_napiecie[2] > 9.9 THEN
	    // błąd pomiaru (przerwa w obwodzie) ustaw 0
	    "dbtags_Sterowanie"."Analog pomiar".kolman_poziom_zbiornik_3 := 0.0;
	  ELSE
	    // pomiar ok
	    "dbtags_Sterowanie"."Analog pomiar".kolman_poziom_zbiornik_3 := (100 * "KALMAN_DB".kalman_napiecie[2]);
	    ;
	  END_IF;
	  // zbiornik 4
	  IF "KALMAN_DB".kalman_napiecie[3] > 9.9 THEN
	    // błąd pomiaru (przerwa w obwodzie) ustaw 0
	    "dbtags_Sterowanie"."Analog pomiar".kolman_poziom_zbiornik_4 := 0.0;
	  ELSE
	    // pomiar ok
	    "dbtags_Sterowanie"."Analog pomiar".kolman_poziom_zbiornik_4 := (100 * "KALMAN_DB".kalman_napiecie[3]);
	    ;
	  END_IF;
	  
	  // Ciśnienie B5 magistrala
	  IF "KALMAN_DB".kalman_napiecie[4] >= 23.0 THEN
	    //błąd pomiaru ustawienie max 
	    "dbtags_Sterowanie"."Analog pomiar".ciśnienie_B5 := 0.0;
	  ELSE
	    // pomiar ok
	    "dbtags_Sterowanie"."Analog pomiar".ciśnienie_B5 := "KALMAN_DB".kalman_napiecie[4];
	    ;
	  END_IF;
	  
	  
	END_REGION
	
	
	REGION Przepływomierz
	  // Konwersja i skalowanie
	  "dbdane".Wielkość_przepływu_Q2_analog := "SclScaleLinearIntToReal"(x := "AI_przepływ",
	                                                                    yMin := "Parametryzacja"."Setting analog".minPrzepływomierz_Q2,
	                                                                    yMax := "Parametryzacja"."Setting analog".maxPrzepływomierz_Q2,
	                                                                    y0 := "Parametryzacja"."Setting analog".minPrzepływomierz_Q2,
	                                                                    x0 := 0, x1 := 27648,
	                                                                    y1 := "Parametryzacja"."Setting analog".maxPrzepływomierz_Q2);
	END_REGION
	
	REGION Ciśnienie B5
	  // Konwersja i skalowanie
	  "dbtags_Sterowanie"."Analog pomiar".AI_ciśnienie_B5 := "SclScaleLinearIntToReal"(x := "AI_ciśnienie_B5",
	                                                                                 yMin := "Parametryzacja"."Setting analog".minPrzetwornikCiśnienia_B5,
	                                                                                 yMax := "Parametryzacja"."Setting analog".maxPrzetwornikCiśnienia_B5,
	                                                                                 y0 := "Parametryzacja"."Setting analog".minPrzetwornikCiśnienia_B5,
	                                                                                 x0 := 0,
	                                                                                 x1 := 27648,
	                                                                                 y1 := "Parametryzacja"."Setting analog".maxPrzetwornikCiśnienia_B5);
	END_REGION
	
	
	REGION Poziom w zbiornikach 
	  // Konwersja i skalowanie pomiarów z wejść analogowych
	  // Zbiornik 1
	  "dbtags_Sterowanie"."Analog pomiar".AI_poziom_zbiornik_1 := "SclScaleLinearIntToReal"(x := "AI_poziom_zbiornik_1",
	                                                                         yMin := "Parametryzacja"."Setting analog".minSondaHydro,
	                                                                         yMax := "Parametryzacja"."Setting analog".maxSondaHydro,
	                                                                         y0 := "Parametryzacja"."Setting analog".minSondaHydro,
	                                                                         x0 := 0,
	                                                                         x1 := 27648,
	                                                                         y1 := "Parametryzacja"."Setting analog".maxSondaHydro);
	  
	  // Zbiornik 2
	"dbtags_Sterowanie"."Analog pomiar".AI_poziom_zbiornik_2 := "SclScaleLinearIntToReal"(x := "AI_poziom_zbiornik_2",
	                                                                         yMin := "Parametryzacja"."Setting analog".minSondaHydro,
	                                                                         yMax := "Parametryzacja"."Setting analog".maxSondaHydro,
	                                                                         y0 := "Parametryzacja"."Setting analog".minSondaHydro,
	                                                                         x0 := 0,
	                                                                         x1 := 27648,
	                                                                         y1 := "Parametryzacja"."Setting analog".maxSondaHydro);
	  
	  // Zbiornik 3
	"dbtags_Sterowanie"."Analog pomiar".AI_poziom_zbiornik_3 := "SclScaleLinearIntToReal"(x := "AI_poziom_zbiornik_3",
	                                                                         yMin := "Parametryzacja"."Setting analog".minSondaHydro,
	                                                                         yMax := "Parametryzacja"."Setting analog".maxSondaHydro,
	                                                                         y0 := "Parametryzacja"."Setting analog".minSondaHydro,
	                                                                         x0 := 0,
	                                                                         x1 := 27648,
	                                                                         y1 := "Parametryzacja"."Setting analog".maxSondaHydro);
	  
	  // Zbiornik 4
	"dbtags_Sterowanie"."Analog pomiar".AI_poziom_zbiornik_4 := "SclScaleLinearIntToReal"(x := "AI_poziom_zbiornik_4",
	                                                                         yMin := "Parametryzacja"."Setting analog".minSondaHydro,
	                                                                         yMax := "Parametryzacja"."Setting analog".maxSondaHydro,
	                                                                         y0 := "Parametryzacja"."Setting analog".minSondaHydro,
	                                                                         x0 := 0,
	                                                                         x1 := 27648,
	                                                                         y1 := "Parametryzacja"."Setting analog".maxSondaHydro);
	  
	END_REGION
	
	
	
	
	
	
	
	
	
	
	
	
	
	
	
	
	
	
	
	
	
END_FUNCTION

FUNCTION "Gotowość_i_Sygnalizacja" : Void   // FC8, LAD
TITLE = Ustawienie Gotowośći
{ S7_Optimized_Access := 'TRUE' }
AUTHOR : rtecmer
VERSION : 0.1
// Funkcja w zależności od przełącznika technologiczne związanego z przebudową zasuw z Czeskich na AUMA przełącza sygnał godowości w zależności jak ajest zasuwa podłączona w procesie technologicznym
// stored: AutoNumber true, IsIECCheckEnabled false, SetENOAutomatically false, UDAEnableTagReadback false
   VAR_TEMP   // added for the SCL form of the ladder/FBD networks
      _w1 : Bool;
   END_VAR
BEGIN

REGION Network 1 (SCL): Pływaki minimum - Zbiorniki Zb1 - 4
   // min pływak
   "Zmienne_sterujące_zbiorników".Zbiornik_1.is_min_float_Zb := "float_min_tank_1";
   "Zmienne_sterujące_zbiorników".Zbiornik_2.is_min_float_Zb := "float_min_tank_2";
   "Zmienne_sterujące_zbiorników".Zbiornik_3.is_min_float_Zb := "float_min_tank_3";
   "Zmienne_sterujące_zbiorników".Zbiornik_4.is_min_float_Zb := "float_min_tank_4";
   // max pływak
   "Zmienne_sterujące_zbiorników".Zbiornik_1.is_max_float_Zb := "float_max_tank_1";
   "Zmienne_sterujące_zbiorników".Zbiornik_2.is_max_float_Zb := "float_max_tank_2";
   "Zmienne_sterujące_zbiorników".Zbiornik_3.is_max_float_Zb := "float_max_tank_3";
   "Zmienne_sterujące_zbiorników".Zbiornik_4.is_max_float_Zb := "float_max_tank_4";
END_REGION

REGION Network 2: bit gotowości wspólny Z10
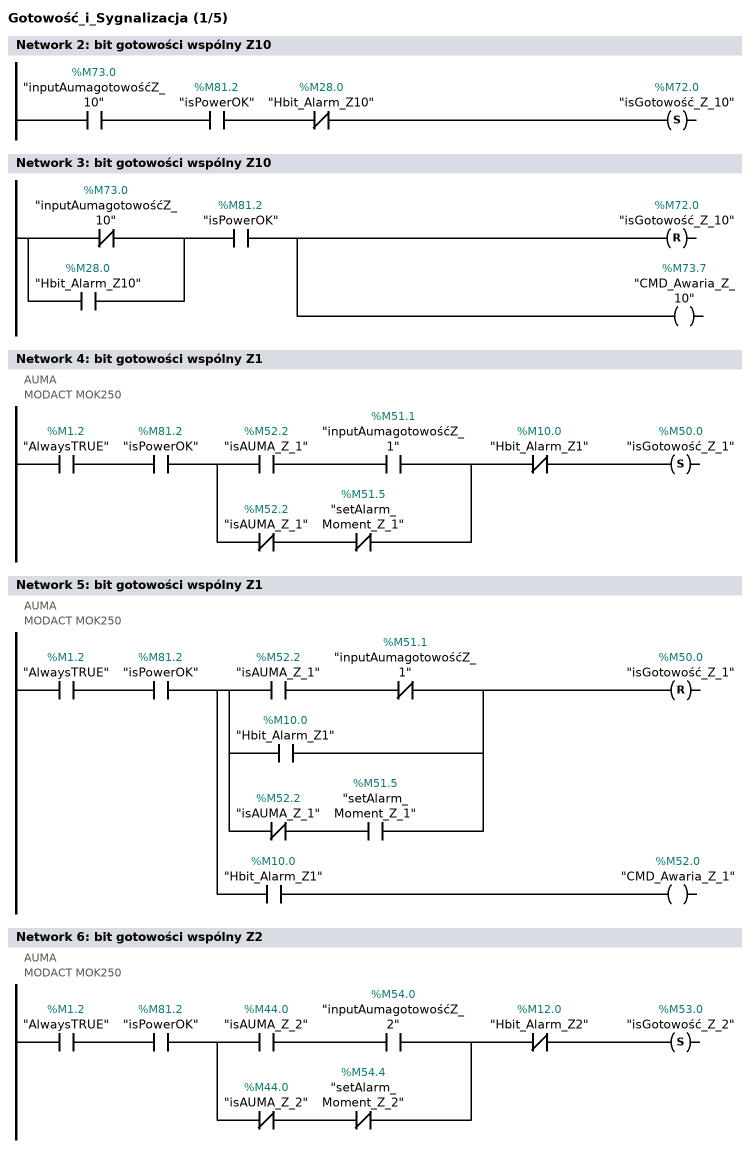
   RUNG wire#powerrail
      Contact( "inputAumagotowośćZ_10" )
      Contact( "isPowerOK" )
      I_Contact( "Hbit_Alarm_Z10" )
      S_Coil( "isGotowość_Z_10" )
   END_RUNG
   // the same network as SCL:
   IF "inputAumagotowośćZ_10" AND "isPowerOK" AND NOT "Hbit_Alarm_Z10" THEN
       "isGotowość_Z_10" := TRUE;
   END_IF;
END_REGION

REGION Network 3: bit gotowości wspólny Z10
   RUNG wire#powerrail
      I_Contact( "inputAumagotowośćZ_10" )
      wire#w1
      Contact( "isPowerOK" )
      wire#w2
      R_Coil( "isGotowość_Z_10" )
   END_RUNG
   RUNG wire#powerrail
      Contact( "Hbit_Alarm_Z10" )
   END_RUNG wire#w1
   RUNG wire#w2
      Coil( "CMD_Awaria_Z_10" )
   END_RUNG
   // the same network as SCL:
   #_w1 := (NOT "inputAumagotowośćZ_10" OR "Hbit_Alarm_Z10") AND "isPowerOK";
   IF #_w1 THEN "isGotowość_Z_10" := FALSE; END_IF;
   "CMD_Awaria_Z_10" := #_w1;
END_REGION

REGION Network 4: bit gotowości wspólny Z1
   // AUMA
   // MODACT MOK250
   RUNG wire#powerrail
      Contact( "AlwaysTRUE" )
      Contact( "isPowerOK" )
      wire#w1
      Contact( "isAUMA_Z_1" )
      Contact( "inputAumagotowośćZ_1" )
      wire#w2
      I_Contact( "Hbit_Alarm_Z1" )
      S_Coil( "isGotowość_Z_1" )
   END_RUNG
   RUNG wire#w1
      I_Contact( "isAUMA_Z_1" )
      I_Contact( "setAlarm_Moment_Z_1" )
   END_RUNG wire#w2
   // the same network as SCL:
   IF "AlwaysTRUE" AND "isPowerOK" AND (("isAUMA_Z_1" AND "inputAumagotowośćZ_1") OR (NOT "isAUMA_Z_1" AND NOT "setAlarm_Moment_Z_1")) AND NOT "Hbit_Alarm_Z1" THEN
       "isGotowość_Z_1" := TRUE;
   END_IF;
END_REGION

REGION Network 5: bit gotowości wspólny Z1
   // AUMA
   // MODACT MOK250
   RUNG wire#powerrail
      Contact( "AlwaysTRUE" )
      Contact( "isPowerOK" )
      wire#w1
      Contact( "isAUMA_Z_1" )
      I_Contact( "inputAumagotowośćZ_1" )
      wire#w2
      R_Coil( "isGotowość_Z_1" )
   END_RUNG
   RUNG wire#w1
      Contact( "Hbit_Alarm_Z1" )
   END_RUNG wire#w2
   RUNG wire#w1
      I_Contact( "isAUMA_Z_1" )
      Contact( "setAlarm_Moment_Z_1" )
   END_RUNG wire#w2
   RUNG wire#w1
      Contact( "Hbit_Alarm_Z1" )
      Coil( "CMD_Awaria_Z_1" )
   END_RUNG
   // the same network as SCL:
   #_w1 := "AlwaysTRUE" AND "isPowerOK";
   IF #_w1 AND (("isAUMA_Z_1" AND NOT "inputAumagotowośćZ_1") OR "Hbit_Alarm_Z1" OR (NOT "isAUMA_Z_1" AND "setAlarm_Moment_Z_1")) THEN
       "isGotowość_Z_1" := FALSE;
   END_IF;
   "CMD_Awaria_Z_1" := #_w1 AND "Hbit_Alarm_Z1";
END_REGION

REGION Network 6: bit gotowości wspólny Z2
   // AUMA
   // MODACT MOK250
   RUNG wire#powerrail
      Contact( "AlwaysTRUE" )
      Contact( "isPowerOK" )
      wire#w1
      Contact( "isAUMA_Z_2" )
      Contact( "inputAumagotowośćZ_2" )
      wire#w2
      I_Contact( "Hbit_Alarm_Z2" )
      S_Coil( "isGotowość_Z_2" )
   END_RUNG
   RUNG wire#w1
      I_Contact( "isAUMA_Z_2" )
      I_Contact( "setAlarm_Moment_Z_2" )
   END_RUNG wire#w2
   // the same network as SCL:
   IF "AlwaysTRUE" AND "isPowerOK" AND (("isAUMA_Z_2" AND "inputAumagotowośćZ_2") OR (NOT "isAUMA_Z_2" AND NOT "setAlarm_Moment_Z_2")) AND NOT "Hbit_Alarm_Z2" THEN
       "isGotowość_Z_2" := TRUE;
   END_IF;
END_REGION

REGION Network 7: bit gotowości wspólny Z2
   // AUMA
   // MODACT MOK250
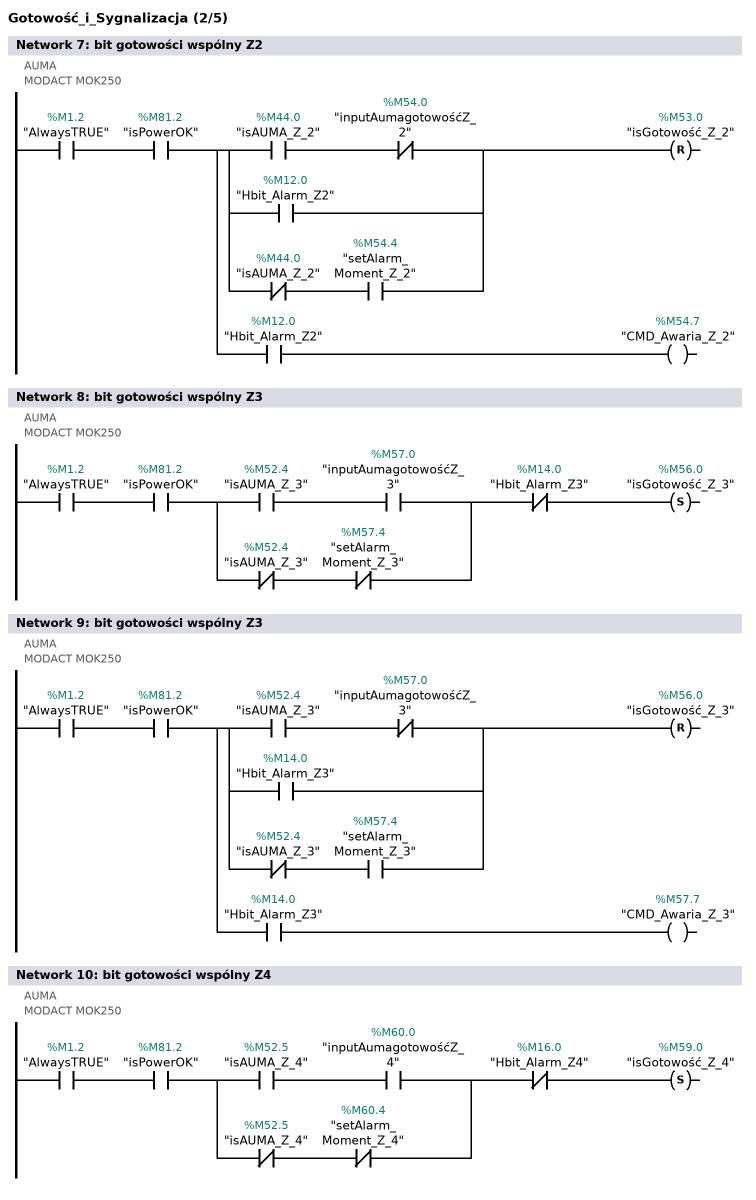
   RUNG wire#powerrail
      Contact( "AlwaysTRUE" )
      Contact( "isPowerOK" )
      wire#w1
      Contact( "isAUMA_Z_2" )
      I_Contact( "inputAumagotowośćZ_2" )
      wire#w2
      R_Coil( "isGotowość_Z_2" )
   END_RUNG
   RUNG wire#w1
      Contact( "Hbit_Alarm_Z2" )
   END_RUNG wire#w2
   RUNG wire#w1
      I_Contact( "isAUMA_Z_2" )
      Contact( "setAlarm_Moment_Z_2" )
   END_RUNG wire#w2
   RUNG wire#w1
      Contact( "Hbit_Alarm_Z2" )
      Coil( "CMD_Awaria_Z_2" )
   END_RUNG
   // the same network as SCL:
   #_w1 := "AlwaysTRUE" AND "isPowerOK";
   IF #_w1 AND (("isAUMA_Z_2" AND NOT "inputAumagotowośćZ_2") OR "Hbit_Alarm_Z2" OR (NOT "isAUMA_Z_2" AND "setAlarm_Moment_Z_2")) THEN
       "isGotowość_Z_2" := FALSE;
   END_IF;
   "CMD_Awaria_Z_2" := #_w1 AND "Hbit_Alarm_Z2";
END_REGION

REGION Network 8: bit gotowości wspólny Z3
   // AUMA
   // MODACT MOK250
   RUNG wire#powerrail
      Contact( "AlwaysTRUE" )
      Contact( "isPowerOK" )
      wire#w1
      Contact( "isAUMA_Z_3" )
      Contact( "inputAumagotowośćZ_3" )
      wire#w2
      I_Contact( "Hbit_Alarm_Z3" )
      S_Coil( "isGotowość_Z_3" )
   END_RUNG
   RUNG wire#w1
      I_Contact( "isAUMA_Z_3" )
      I_Contact( "setAlarm_Moment_Z_3" )
   END_RUNG wire#w2
   // the same network as SCL:
   IF "AlwaysTRUE" AND "isPowerOK" AND (("isAUMA_Z_3" AND "inputAumagotowośćZ_3") OR (NOT "isAUMA_Z_3" AND NOT "setAlarm_Moment_Z_3")) AND NOT "Hbit_Alarm_Z3" THEN
       "isGotowość_Z_3" := TRUE;
   END_IF;
END_REGION

REGION Network 9: bit gotowości wspólny Z3
   // AUMA
   // MODACT MOK250
   RUNG wire#powerrail
      Contact( "AlwaysTRUE" )
      Contact( "isPowerOK" )
      wire#w1
      Contact( "isAUMA_Z_3" )
      I_Contact( "inputAumagotowośćZ_3" )
      wire#w2
      R_Coil( "isGotowość_Z_3" )
   END_RUNG
   RUNG wire#w1
      Contact( "Hbit_Alarm_Z3" )
   END_RUNG wire#w2
   RUNG wire#w1
      I_Contact( "isAUMA_Z_3" )
      Contact( "setAlarm_Moment_Z_3" )
   END_RUNG wire#w2
   RUNG wire#w1
      Contact( "Hbit_Alarm_Z3" )
      Coil( "CMD_Awaria_Z_3" )
   END_RUNG
   // the same network as SCL:
   #_w1 := "AlwaysTRUE" AND "isPowerOK";
   IF #_w1 AND (("isAUMA_Z_3" AND NOT "inputAumagotowośćZ_3") OR "Hbit_Alarm_Z3" OR (NOT "isAUMA_Z_3" AND "setAlarm_Moment_Z_3")) THEN
       "isGotowość_Z_3" := FALSE;
   END_IF;
   "CMD_Awaria_Z_3" := #_w1 AND "Hbit_Alarm_Z3";
END_REGION

REGION Network 10: bit gotowości wspólny Z4
   // AUMA
   // MODACT MOK250
   RUNG wire#powerrail
      Contact( "AlwaysTRUE" )
      Contact( "isPowerOK" )
      wire#w1
      Contact( "isAUMA_Z_4" )
      Contact( "inputAumagotowośćZ_4" )
      wire#w2
      I_Contact( "Hbit_Alarm_Z4" )
      S_Coil( "isGotowość_Z_4" )
   END_RUNG
   RUNG wire#w1
      I_Contact( "isAUMA_Z_4" )
      I_Contact( "setAlarm_Moment_Z_4" )
   END_RUNG wire#w2
   // the same network as SCL:
   IF "AlwaysTRUE" AND "isPowerOK" AND (("isAUMA_Z_4" AND "inputAumagotowośćZ_4") OR (NOT "isAUMA_Z_4" AND NOT "setAlarm_Moment_Z_4")) AND NOT "Hbit_Alarm_Z4" THEN
       "isGotowość_Z_4" := TRUE;
   END_IF;
END_REGION

REGION Network 11: bit gotowości wspólny Z4
   // AUMA
   // MODACT MOK250
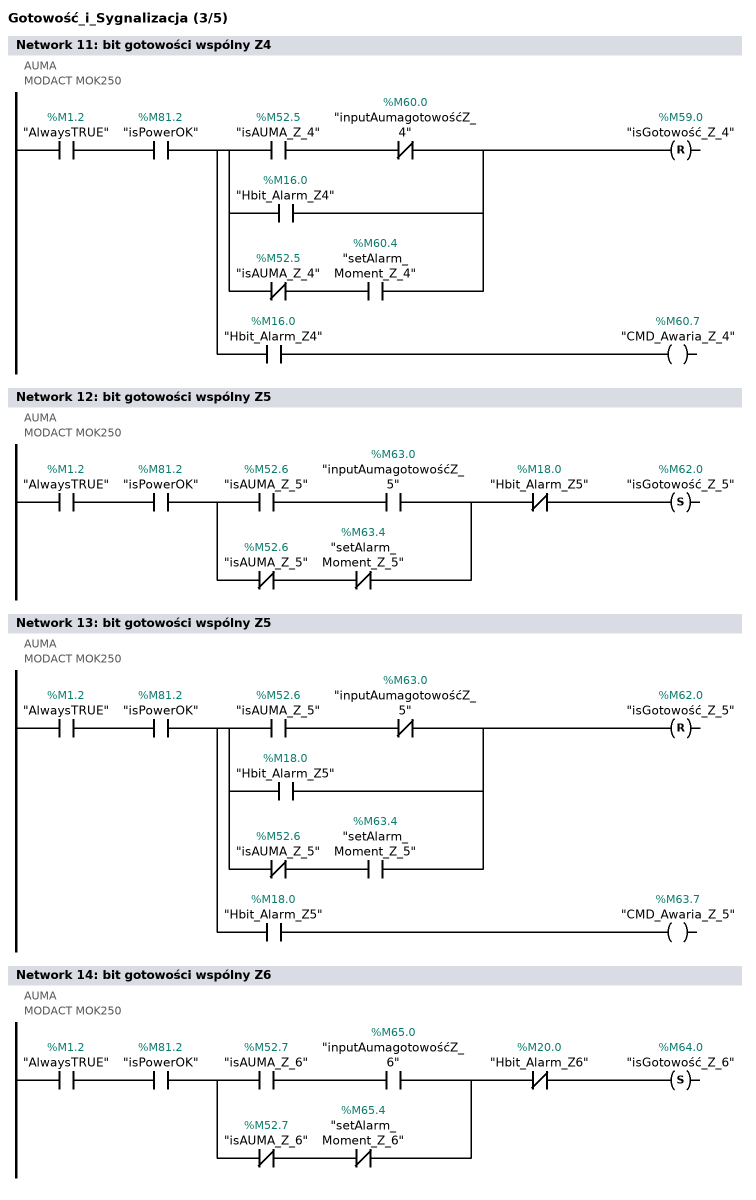
   RUNG wire#powerrail
      Contact( "AlwaysTRUE" )
      Contact( "isPowerOK" )
      wire#w1
      Contact( "isAUMA_Z_4" )
      I_Contact( "inputAumagotowośćZ_4" )
      wire#w2
      R_Coil( "isGotowość_Z_4" )
   END_RUNG
   RUNG wire#w1
      Contact( "Hbit_Alarm_Z4" )
   END_RUNG wire#w2
   RUNG wire#w1
      I_Contact( "isAUMA_Z_4" )
      Contact( "setAlarm_Moment_Z_4" )
   END_RUNG wire#w2
   RUNG wire#w1
      Contact( "Hbit_Alarm_Z4" )
      Coil( "CMD_Awaria_Z_4" )
   END_RUNG
   // the same network as SCL:
   #_w1 := "AlwaysTRUE" AND "isPowerOK";
   IF #_w1 AND (("isAUMA_Z_4" AND NOT "inputAumagotowośćZ_4") OR "Hbit_Alarm_Z4" OR (NOT "isAUMA_Z_4" AND "setAlarm_Moment_Z_4")) THEN
       "isGotowość_Z_4" := FALSE;
   END_IF;
   "CMD_Awaria_Z_4" := #_w1 AND "Hbit_Alarm_Z4";
END_REGION

REGION Network 12: bit gotowości wspólny Z5
   // AUMA
   // MODACT MOK250
   RUNG wire#powerrail
      Contact( "AlwaysTRUE" )
      Contact( "isPowerOK" )
      wire#w1
      Contact( "isAUMA_Z_5" )
      Contact( "inputAumagotowośćZ_5" )
      wire#w2
      I_Contact( "Hbit_Alarm_Z5" )
      S_Coil( "isGotowość_Z_5" )
   END_RUNG
   RUNG wire#w1
      I_Contact( "isAUMA_Z_5" )
      I_Contact( "setAlarm_Moment_Z_5" )
   END_RUNG wire#w2
   // the same network as SCL:
   IF "AlwaysTRUE" AND "isPowerOK" AND (("isAUMA_Z_5" AND "inputAumagotowośćZ_5") OR (NOT "isAUMA_Z_5" AND NOT "setAlarm_Moment_Z_5")) AND NOT "Hbit_Alarm_Z5" THEN
       "isGotowość_Z_5" := TRUE;
   END_IF;
END_REGION

REGION Network 13: bit gotowości wspólny Z5
   // AUMA
   // MODACT MOK250
   RUNG wire#powerrail
      Contact( "AlwaysTRUE" )
      Contact( "isPowerOK" )
      wire#w1
      Contact( "isAUMA_Z_5" )
      I_Contact( "inputAumagotowośćZ_5" )
      wire#w2
      R_Coil( "isGotowość_Z_5" )
   END_RUNG
   RUNG wire#w1
      Contact( "Hbit_Alarm_Z5" )
   END_RUNG wire#w2
   RUNG wire#w1
      I_Contact( "isAUMA_Z_5" )
      Contact( "setAlarm_Moment_Z_5" )
   END_RUNG wire#w2
   RUNG wire#w1
      Contact( "Hbit_Alarm_Z5" )
      Coil( "CMD_Awaria_Z_5" )
   END_RUNG
   // the same network as SCL:
   #_w1 := "AlwaysTRUE" AND "isPowerOK";
   IF #_w1 AND (("isAUMA_Z_5" AND NOT "inputAumagotowośćZ_5") OR "Hbit_Alarm_Z5" OR (NOT "isAUMA_Z_5" AND "setAlarm_Moment_Z_5")) THEN
       "isGotowość_Z_5" := FALSE;
   END_IF;
   "CMD_Awaria_Z_5" := #_w1 AND "Hbit_Alarm_Z5";
END_REGION

REGION Network 14: bit gotowości wspólny Z6
   // AUMA
   // MODACT MOK250
   RUNG wire#powerrail
      Contact( "AlwaysTRUE" )
      Contact( "isPowerOK" )
      wire#w1
      Contact( "isAUMA_Z_6" )
      Contact( "inputAumagotowośćZ_6" )
      wire#w2
      I_Contact( "Hbit_Alarm_Z6" )
      S_Coil( "isGotowość_Z_6" )
   END_RUNG
   RUNG wire#w1
      I_Contact( "isAUMA_Z_6" )
      I_Contact( "setAlarm_Moment_Z_6" )
   END_RUNG wire#w2
   // the same network as SCL:
   IF "AlwaysTRUE" AND "isPowerOK" AND (("isAUMA_Z_6" AND "inputAumagotowośćZ_6") OR (NOT "isAUMA_Z_6" AND NOT "setAlarm_Moment_Z_6")) AND NOT "Hbit_Alarm_Z6" THEN
       "isGotowość_Z_6" := TRUE;
   END_IF;
END_REGION

REGION Network 15: bit gotowości wspólny Z6
   // AUMA
   // MODACT MOK250
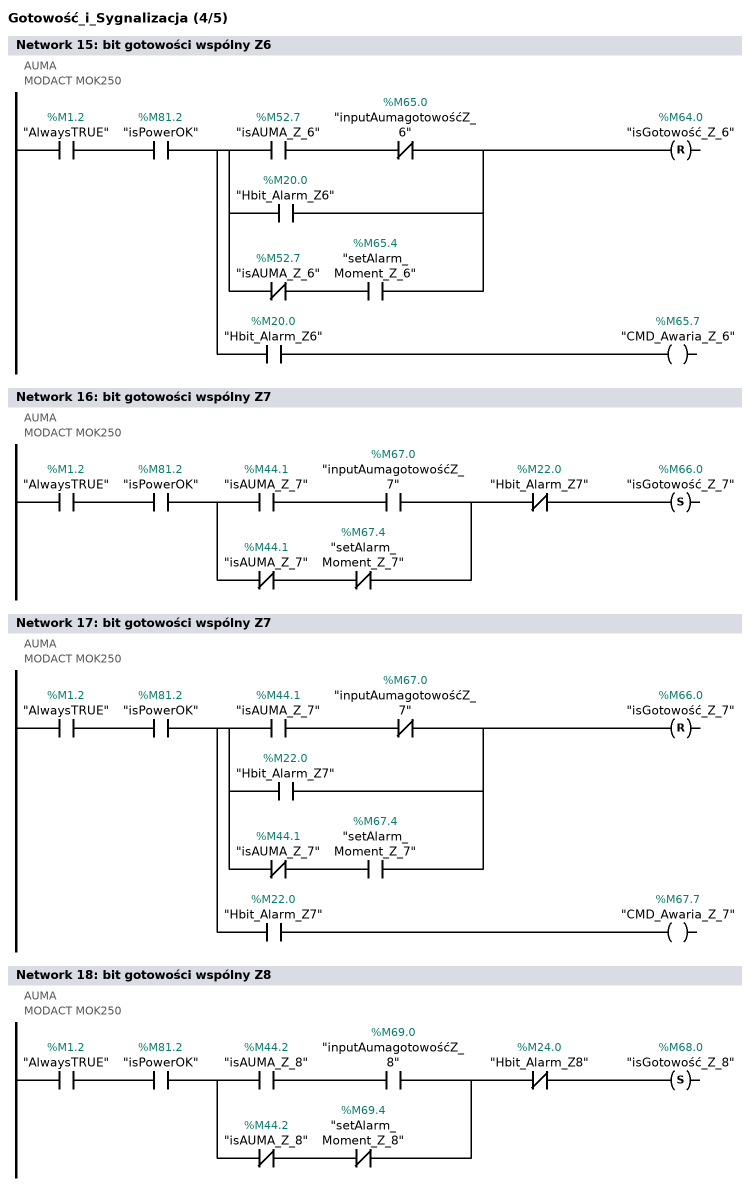
   RUNG wire#powerrail
      Contact( "AlwaysTRUE" )
      Contact( "isPowerOK" )
      wire#w1
      Contact( "isAUMA_Z_6" )
      I_Contact( "inputAumagotowośćZ_6" )
      wire#w2
      R_Coil( "isGotowość_Z_6" )
   END_RUNG
   RUNG wire#w1
      Contact( "Hbit_Alarm_Z6" )
   END_RUNG wire#w2
   RUNG wire#w1
      I_Contact( "isAUMA_Z_6" )
      Contact( "setAlarm_Moment_Z_6" )
   END_RUNG wire#w2
   RUNG wire#w1
      Contact( "Hbit_Alarm_Z6" )
      Coil( "CMD_Awaria_Z_6" )
   END_RUNG
   // the same network as SCL:
   #_w1 := "AlwaysTRUE" AND "isPowerOK";
   IF #_w1 AND (("isAUMA_Z_6" AND NOT "inputAumagotowośćZ_6") OR "Hbit_Alarm_Z6" OR (NOT "isAUMA_Z_6" AND "setAlarm_Moment_Z_6")) THEN
       "isGotowość_Z_6" := FALSE;
   END_IF;
   "CMD_Awaria_Z_6" := #_w1 AND "Hbit_Alarm_Z6";
END_REGION

REGION Network 16: bit gotowości wspólny Z7
   // AUMA
   // MODACT MOK250
   RUNG wire#powerrail
      Contact( "AlwaysTRUE" )
      Contact( "isPowerOK" )
      wire#w1
      Contact( "isAUMA_Z_7" )
      Contact( "inputAumagotowośćZ_7" )
      wire#w2
      I_Contact( "Hbit_Alarm_Z7" )
      S_Coil( "isGotowość_Z_7" )
   END_RUNG
   RUNG wire#w1
      I_Contact( "isAUMA_Z_7" )
      I_Contact( "setAlarm_Moment_Z_7" )
   END_RUNG wire#w2
   // the same network as SCL:
   IF "AlwaysTRUE" AND "isPowerOK" AND (("isAUMA_Z_7" AND "inputAumagotowośćZ_7") OR (NOT "isAUMA_Z_7" AND NOT "setAlarm_Moment_Z_7")) AND NOT "Hbit_Alarm_Z7" THEN
       "isGotowość_Z_7" := TRUE;
   END_IF;
END_REGION

REGION Network 17: bit gotowości wspólny Z7
   // AUMA
   // MODACT MOK250
   RUNG wire#powerrail
      Contact( "AlwaysTRUE" )
      Contact( "isPowerOK" )
      wire#w1
      Contact( "isAUMA_Z_7" )
      I_Contact( "inputAumagotowośćZ_7" )
      wire#w2
      R_Coil( "isGotowość_Z_7" )
   END_RUNG
   RUNG wire#w1
      Contact( "Hbit_Alarm_Z7" )
   END_RUNG wire#w2
   RUNG wire#w1
      I_Contact( "isAUMA_Z_7" )
      Contact( "setAlarm_Moment_Z_7" )
   END_RUNG wire#w2
   RUNG wire#w1
      Contact( "Hbit_Alarm_Z7" )
      Coil( "CMD_Awaria_Z_7" )
   END_RUNG
   // the same network as SCL:
   #_w1 := "AlwaysTRUE" AND "isPowerOK";
   IF #_w1 AND (("isAUMA_Z_7" AND NOT "inputAumagotowośćZ_7") OR "Hbit_Alarm_Z7" OR (NOT "isAUMA_Z_7" AND "setAlarm_Moment_Z_7")) THEN
       "isGotowość_Z_7" := FALSE;
   END_IF;
   "CMD_Awaria_Z_7" := #_w1 AND "Hbit_Alarm_Z7";
END_REGION

REGION Network 18: bit gotowości wspólny Z8
   // AUMA
   // MODACT MOK250
   RUNG wire#powerrail
      Contact( "AlwaysTRUE" )
      Contact( "isPowerOK" )
      wire#w1
      Contact( "isAUMA_Z_8" )
      Contact( "inputAumagotowośćZ_8" )
      wire#w2
      I_Contact( "Hbit_Alarm_Z8" )
      S_Coil( "isGotowość_Z_8" )
   END_RUNG
   RUNG wire#w1
      I_Contact( "isAUMA_Z_8" )
      I_Contact( "setAlarm_Moment_Z_8" )
   END_RUNG wire#w2
   // the same network as SCL:
   IF "AlwaysTRUE" AND "isPowerOK" AND (("isAUMA_Z_8" AND "inputAumagotowośćZ_8") OR (NOT "isAUMA_Z_8" AND NOT "setAlarm_Moment_Z_8")) AND NOT "Hbit_Alarm_Z8" THEN
       "isGotowość_Z_8" := TRUE;
   END_IF;
END_REGION

REGION Network 19: bit gotowości wspólny Z8
   // AUMA
   // MODACT MOK250
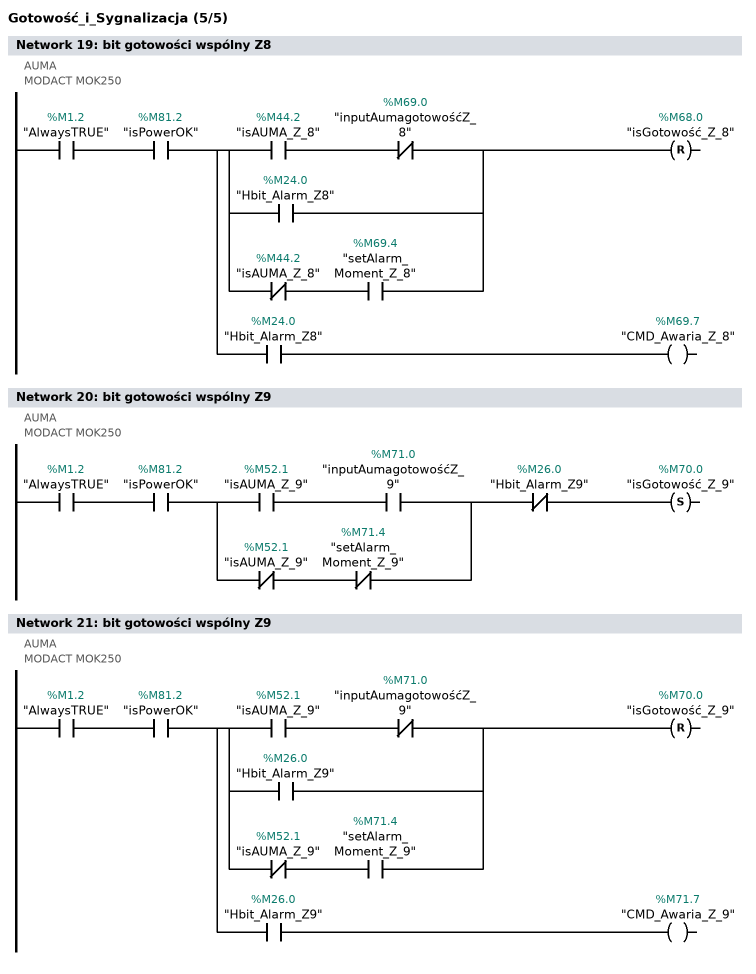
   RUNG wire#powerrail
      Contact( "AlwaysTRUE" )
      Contact( "isPowerOK" )
      wire#w1
      Contact( "isAUMA_Z_8" )
      I_Contact( "inputAumagotowośćZ_8" )
      wire#w2
      R_Coil( "isGotowość_Z_8" )
   END_RUNG
   RUNG wire#w1
      Contact( "Hbit_Alarm_Z8" )
   END_RUNG wire#w2
   RUNG wire#w1
      I_Contact( "isAUMA_Z_8" )
      Contact( "setAlarm_Moment_Z_8" )
   END_RUNG wire#w2
   RUNG wire#w1
      Contact( "Hbit_Alarm_Z8" )
      Coil( "CMD_Awaria_Z_8" )
   END_RUNG
   // the same network as SCL:
   #_w1 := "AlwaysTRUE" AND "isPowerOK";
   IF #_w1 AND (("isAUMA_Z_8" AND NOT "inputAumagotowośćZ_8") OR "Hbit_Alarm_Z8" OR (NOT "isAUMA_Z_8" AND "setAlarm_Moment_Z_8")) THEN
       "isGotowość_Z_8" := FALSE;
   END_IF;
   "CMD_Awaria_Z_8" := #_w1 AND "Hbit_Alarm_Z8";
END_REGION

REGION Network 20: bit gotowości wspólny Z9
   // AUMA
   // MODACT MOK250
   RUNG wire#powerrail
      Contact( "AlwaysTRUE" )
      Contact( "isPowerOK" )
      wire#w1
      Contact( "isAUMA_Z_9" )
      Contact( "inputAumagotowośćZ_9" )
      wire#w2
      I_Contact( "Hbit_Alarm_Z9" )
      S_Coil( "isGotowość_Z_9" )
   END_RUNG
   RUNG wire#w1
      I_Contact( "isAUMA_Z_9" )
      I_Contact( "setAlarm_Moment_Z_9" )
   END_RUNG wire#w2
   // the same network as SCL:
   IF "AlwaysTRUE" AND "isPowerOK" AND (("isAUMA_Z_9" AND "inputAumagotowośćZ_9") OR (NOT "isAUMA_Z_9" AND NOT "setAlarm_Moment_Z_9")) AND NOT "Hbit_Alarm_Z9" THEN
       "isGotowość_Z_9" := TRUE;
   END_IF;
END_REGION

